# B&R Automation Studio project NAEUL004C00R13L518F00 (part 75)

#### PrecededBySelfBackground1.st
```iecst
ACTION PrecededBySelfBackground1:

	//Converting BA from US Hermes to Rcp
	IF p_bLinkOpsRun THEN
		IF  p_bHermesBADataAccepted THEN
			tyCurrReqRcp.sBoardId := p_tyHermesBARcv.tyData.sBoardId;
			tyCurrReqRcp.sBoardIdCreatedBy := p_tyHermesBARcv.tyData.sBoardIdCreatedBy;
			tyCurrReqRcp.eFailedBoard := p_tyHermesBARcv.tyData.eFailedBoard;
			tyCurrReqRcp.sProductTypeId := p_tyHermesBARcv.tyData.sProductTypeId;
			tyCurrReqRcp.eFlippedBoard := p_tyHermesBARcv.tyData.eFlippedBoard;
			tyCurrReqRcp.sTopBarcode := p_tyHermesBARcv.tyData.sTopBarcode;
			tyCurrReqRcp.sBottomBarcode := p_tyHermesBARcv.tyData.sBottomBarcode;
			tyCurrReqRcp.rLength := p_tyHermesBARcv.tyData.rLength;
			tyCurrReqRcp.rWidth := p_tyHermesBARcv.tyData.rWidth;
			tyCurrReqRcp.rThickness := p_tyHermesBARcv.tyData.rThickness;
			tyCurrReqRcp.rConveyorSpeed := p_tyHermesBARcv.tyData.rConveyorSpeed;
			tyCurrReqRcp.rTopClearanceHeight := p_tyHermesBARcv.tyData.rTopClearanceHeight;
			tyCurrReqRcp.rBottomClearanceHeight := p_tyHermesBARcv.tyData.rBottomClearanceHeight;
			tyCurrReqRcp.rWeight := p_tyHermesBARcv.tyData.rWeight;
			tyCurrReqRcp.sWorkOrderId := p_tyHermesBARcv.tyData.sWorkOrderId;
			tyCurrReqRcp.sBatchId := p_tyHermesBARcv.tyData.sBatchId;
		ELSIF p_bHermesBFDataAccepted THEN
			//Converting BF from US Hermes to Rcp
			tyCurrReqRcp.sBoardId := p_tyHermesBFRcv.tyData.sBoardId;
			tyCurrReqRcp.sBoardIdCreatedBy := p_tyHermesBFRcv.tyData.sBoardIdCreatedBy;
			tyCurrReqRcp.eFailedBoard := p_tyHermesBFRcv.tyData.eFailedBoard;
			tyCurrReqRcp.sProductTypeId := p_tyHermesBFRcv.tyData.sProductTypeId;
			tyCurrReqRcp.eFlippedBoard := p_tyHermesBFRcv.tyData.eFlippedBoard;
			tyCurrReqRcp.sTopBarcode := p_tyHermesBFRcv.tyData.sTopBarcode;
			tyCurrReqRcp.sBottomBarcode := p_tyHermesBFRcv.tyData.sBottomBarcode;
			tyCurrReqRcp.rLength := p_tyHermesBFRcv.tyData.rLength;
			tyCurrReqRcp.rWidth := p_tyHermesBFRcv.tyData.rWidth;
			tyCurrReqRcp.rThickness := p_tyHermesBFRcv.tyData.rThickness;
			tyCurrReqRcp.rConveyorSpeed := p_tyHermesBFRcv.tyData.rConveyorSpeed;
			tyCurrReqRcp.rTopClearanceHeight := p_tyHermesBFRcv.tyData.rTopClearanceHeight;
			tyCurrReqRcp.rBottomClearanceHeight := p_tyHermesBFRcv.tyData.rBottomClearanceHeight;
			tyCurrReqRcp.rWeight := p_tyHermesBFRcv.tyData.rWeight;
			tyCurrReqRcp.sWorkOrderId := p_tyHermesBFRcv.tyData.sWorkOrderId;
			tyCurrReqRcp.sBatchId := p_tyHermesBFRcv.tyData.sBatchId;
		END_IF
	END_IF

	//For Zone 1 Initialization Only
	IF bInitializedFollower1Done = FALSE AND p_bLinkOpsRun THEN
		IF tyCurrZ1Rcp.rWidth = 0 THEN //nothing found in retain
			IF p_bHermesBrdAvlDataNewBrdAvl1stZ  THEN //if no brd retain
				IF p_tyInternalReqProdRcp.diWidthInUM <> 0 THEN
					tyCurrZ1Rcp.rWidth := p_tyInternalReqProdRcp.diWidthInUM/1000 ;
				ELSE //internalReq Rcp=0
					tyCurrZ1Rcp.rWidth := p_diNtParamProdRcpMinWidth/1000 ;
				END_IF
			ELSE //taken From Hermes Retain
				fbParseBrdAvlExternal.p_XMLTable := ADR(pa_tyLinkXMLTableDataBrdAvl1);
				fbParseBrdAvlExternal.iTotalIdxWrite := p_iLinkXMLTableDataBrdAvlTtlIdx1;
				fbParseBrdAvlExternal;

				tyCurrZ1Rcp.sBoardId := fbParseBrdAvlExternal.tyBoardAvailable.tyData.sBoardId;
				tyCurrZ1Rcp.sBoardIdCreatedBy := fbParseBrdAvlExternal.tyBoardAvailable.tyData.sBoardIdCreatedBy;
				tyCurrZ1Rcp.eFailedBoard := fbParseBrdAvlExternal.tyBoardAvailable.tyData.eFailedBoard;
				tyCurrZ1Rcp.sProductTypeId := fbParseBrdAvlExternal.tyBoardAvailable.tyData.sProductTypeId;
				tyCurrZ1Rcp.eFlippedBoard := fbParseBrdAvlExternal.tyBoardAvailable.tyData.eFlippedBoard;
				tyCurrZ1Rcp.sTopBarcode := fbParseBrdAvlExternal.tyBoardAvailable.tyData.sTopBarcode;
				tyCurrZ1Rcp.sBottomBarcode := fbParseBrdAvlExternal.tyBoardAvailable.tyData.sBottomBarcode;
				tyCurrZ1Rcp.rLength := fbParseBrdAvlExternal.tyBoardAvailable.tyData.rLength;
				tyCurrZ1Rcp.rWidth := fbParseBrdAvlExternal.tyBoardAvailable.tyData.rWidth;
				tyCurrZ1Rcp.rThickness := fbParseBrdAvlExternal.tyBoardAvailable.tyData.rThickness;
				tyCurrZ1Rcp.rConveyorSpeed := fbParseBrdAvlExternal.tyBoardAvailable.tyData.rConveyorSpeed;
				tyCurrZ1Rcp.rTopClearanceHeight := fbParseBrdAvlExternal.tyBoardAvailable.tyData.rTopClearanceHeight;
				tyCurrZ1Rcp.rBottomClearanceHeight := fbParseBrdAvlExternal.tyBoardAvailable.tyData.rBottomClearanceHeight;
				tyCurrZ1Rcp.rWeight := fbParseBrdAvlExternal.tyBoardAvailable.tyData.rWeight;
				tyCurrZ1Rcp.sWorkOrderId := fbParseBrdAvlExternal.tyBoardAvailable.tyData.sWorkOrderId;
				tyCurrZ1Rcp.sBatchId := fbParseBrdAvlExternal.tyBoardAvailable.tyData.sBatchId;
			END_IF
		END_IF
		bOverWriteTravLifProperties := TRUE;
		bInitializedFollower1Done := TRUE;
	END_IF

	//Error Handling
	IF p_bLinkOpsRun AND (p_bHermesBADataAccepted OR p_bHermesBFDataAccepted) THEN //
		IF tyCurrReqRcp.rWidth < DINT_TO_REAL(p_diNtParamProdRcpMinWidth)/1000.0 THEN
			eStatus := Error;
			udiStatus := 10010;
		ELSIF tyCurrReqRcp.rWidth  > DINT_TO_REAL(p_diNtParamProdRcpMaxWidth)/1000.0 THEN
			eStatus := Error;
			udiStatus := 10011;
		ELSIF  tyCurrReqRcp.rThickness  > DINT_TO_REAL(p_eNtParamAutoRcpParamLmt.diThicknessInUM)/1000.0 THEN
			eStatus := Error;
			udiStatus := 10012;
		ELSIF  tyCurrReqRcp.rBottomClearanceHeight  > DINT_TO_REAL(p_eNtParamAutoRcpParamLmt.diMaxBottomCleranceInUM)/1000.0 THEN
			eStatus := Error;
			udiStatus := 10013;
		ELSIF tyCurrReqRcp.rTopClearanceHeight > DINT_TO_REAL(p_eNtParamAutoRcpParamLmt.diMaxTopClearamceInUM)/1000.0 THEN
			eStatus := Error;
			udiStatus := 10014;
		END_IF
		IF eStatus = Error THEN
			memset(ADR(tyCurrReqRcp),0,SIZEOF(tyCurrReqRcp));
		END_IF
	END_IF

	IF eStatus <> Error THEN //do not feed F1 with F2 with invalid recipe
		//Follower1
		IF memcmp(ADR(tyCurrZ1Rcp) , ADR(tyCurrReqRcp) , SIZEOF(tyCurrZ1Rcp)) <> 0 AND tyCurrReqRcp.rWidth <> 0 THEN
			bTravLifWidthDiffBlk := TRUE;
			IF p_bZ1AccNewRcpCondition THEN
				tyCurrZ1Rcp := tyCurrReqRcp;
				bOverWriteTravLifProperties := TRUE;
				usiChg2 := usiChg2 +1;
			END_IF
		ELSE
			bTravLifWidthDiffBlk := FALSE;
			bOverWriteTravLifProperties := TRUE;
		END_IF

		//Follower 2
		FOR ii:= 1 TO SIZEOF(a_bBufferMagPresent)/SIZEOF(a_bBufferMagPresent[1]) DO
			IF p_bZ2AccNewRcpCondition THEN	 //in Ops
				IF a_bBufferMagPresent[ii] = FALSE THEN //all time , at the start time
					memset((ADR(a_tyCurrZ2Rcp[1])+(ii-1)*SIZEOF(a_tyCurrZ2Rcp[1])),0,SIZEOF(a_tyCurrZ2Rcp[1])) ;
					a_bMagChangOverBlk[ii] := FALSE;
				ELSE //if present
					p_tyCmpRcp ACCESS (ADR(a_tyCurrZ2Rcp[1])+(ii-1)*SIZEOF(a_tyCurrZ2Rcp[1])) ;
					a_bCheckDifferent[ii]:= (p_tyCmpRcp.sProductTypeId <> tyCurrZ1Rcp.sProductTypeId) OR
					(p_tyCmpRcp.sBatchId <> tyCurrZ1Rcp.sBatchId AND p_bMcParamAutoRcpBatchIDChgCmp) OR
					(p_tyCmpRcp.sWorkOrderId <> tyCurrZ1Rcp.sWorkOrderId) OR
					p_tyCmpRcp.rWidth <> tyCurrZ1Rcp.rWidth OR
					(p_tyCmpRcp.rTopClearanceHeight <> tyCurrZ1Rcp.rTopClearanceHeight AND NOT(p_bMcParamAutoRcpIgnoreTopClr)) OR
					(p_tyCmpRcp.rBottomClearanceHeight <> tyCurrZ1Rcp.rBottomClearanceHeight AND NOT(p_bMcParamAutoRcpIgnoreBtmClr)) OR
					(p_tyCmpRcp.rThickness <> tyCurrZ1Rcp.rThickness AND NOT(p_bMcParamAutoRcpIgnoreThickns)) OR
					p_tyCmpRcp.eFlippedBoard <> tyCurrZ1Rcp.eFlippedBoard	;
					IF a_bCheckDifferent[ii] THEN
						a_bAllwChangeWidth[ii] := FALSE;
						IF a_tyBffrStat[ii].bBffrMty THEN //udiAllwGo and WidthDiff and empty then change rcp
							p_tyCmpRcp := tyCurrZ1Rcp;
							usiChg := usiChg + 1;
							a_bMagChangOverBlk[ii] := FALSE;
							bOverWriteMagProperties := TRUE;
							a_bAllwChangeSlot[ii]  := TRUE;
						ELSE // WidthDiff and not empty then blk
							a_bMagChangOverBlk[ii] := TRUE;
						END_IF
					ELSE //if rcp same mean changewidth allow change until width is same
						a_bMagChangOverBlk[ii] := FALSE;
						a_bAllwChangeWidth[ii] := (a_bMagAWWidthDiff[ii] OR a_bForceChgWidthIfSameRcp[ii]) AND a_tyBffrStat[ii].bBffrMty AND p_bNtParamProjMagAWPrep;

					END_IF

				END_IF

			END_IF
		END_FOR
	END_IF
	//wait new udiAllwGo to toggle and FIND the other empty to change

	//IF all was block with magazine available then Force the Magazine Exit
	iChgOvrCntr := 0;
	FOR ii:= 1 TO SIZEOF(a_bBufferMagPresent)/SIZEOF(a_bBufferMagPresent[1]) DO
		IF  (a_bBufferMagPresent[ii] AND a_bMagChangOverBlk[ii] = TRUE) THEN
			iChgOvrCntr := iChgOvrCntr +1 ;
			EXIT;
		END_IF
	END_FOR
	IF iChgOvrCntr >= 1 THEN
		bForceExitMag := TRUE; //force Magazine to exit the highest priority Mag
	ELSE
		bForceExitMag := FALSE;
	END_IF

END_ACTION
```

#### PrecededBySelfBackground2.st
```iecst
ACTION PrecededBySelfBackground2:

	//Convert ProdID to Rcp Name and rWidth to diWidth for F0 to output Hermes
	sProdtypeID:= tyCurrReqRcp.sProductTypeId;
	diProdWidth := REAL_TO_DINT(tyCurrReqRcp.rWidth*1000);

	//Convert to Width for F1
	IF bOverWriteTravLifProperties THEN
		diTravLifWidth := REAL_TO_DINT(tyCurrZ1Rcp.rWidth*1000);
		bOverWriteTravLifProperties	:= FALSE;
	END_IF

	//Convert to Pitch for F2
	IF bOverWriteMagProperties = TRUE THEN
		//overwriting diMax
		FOR kk := 1 TO SIZEOF(a_tyCurrZ2Rcp)/SIZEOF(a_tyCurrZ2Rcp[1]) DO
			p_diRequestedMinSlt := 3;
			p_diRequestedGapToMaxSlt := 0;
			IF p_bProdRcp0ToptoBtm THEN
				IF p_diRequestedGapToMaxSlt > ((a_tyCurrZ2Rcp[kk].rTopClearanceHeight + a_tyCurrZ2Rcp[kk].rThickness)/(p_diMagRcpCurrRcpSltToSlt/1000)) THEN
					rMaxslt := (p_diMagRcpCurrRcpTtlSlt-p_diRequestedGapToMaxSlt)  ;
				ELSE
					rMaxslt := p_diMagRcpCurrRcpTtlSlt - ((a_tyCurrZ2Rcp[kk].rTopClearanceHeight + a_tyCurrZ2Rcp[kk].rThickness)/(p_diMagRcpCurrRcpSltToSlt/1000)) + 1;
				END_IF
				rMinslt :=  (a_tyCurrZ2Rcp[kk].rBottomClearanceHeight)/(p_diMagRcpCurrRcpSltToSlt/1000);
				rPitch := (a_tyCurrZ2Rcp[kk].rTopClearanceHeight + a_tyCurrZ2Rcp[kk].rBottomClearanceHeight + a_tyCurrZ2Rcp[kk].rThickness)/(p_diMagRcpCurrRcpSltToSlt/1000);
				IF rPitch = 0 THEN
					rPitch := 1;
				END_IF
				rNumInterval := (rMaxslt - rMinslt )/ceil(rPitch);
				diCalcedMax := REAL_TO_DINT(floor(rMaxslt));
				diCalcedPitch := REAL_TO_DINT(ceil(rPitch));
				diCalcedMin := REAL_TO_DINT((diCalcedMax - floor(rNumInterval)*ceil(rPitch)));

				IF diCalcedMin = 0 THEN
					diCalcedMin := diCalcedPitch;
				END_IF

			ELSE
				IF p_diRequestedMinSlt = 0 THEN
					p_diRequestedMinSlt := 1;
				END_IF
				IF ceil((a_tyCurrZ2Rcp[kk].rBottomClearanceHeight)/(p_diMagRcpCurrRcpSltToSlt/1000)) >= p_diRequestedMinSlt THEN
					rMinslt := (a_tyCurrZ2Rcp[kk].rBottomClearanceHeight)/(p_diMagRcpCurrRcpSltToSlt/1000) + 1;
				ELSE
					rMinslt :=  p_diRequestedMinSlt;
				END_IF
				//+ (a_tyCurrZ2Rcp[kk].rBottomClearanceHeight)/(p_diMagRcpCurrRcpSltToSlt/1000);
				rMaxslt := p_diMagRcpCurrRcpTtlSlt-((a_tyCurrZ2Rcp[kk].rTopClearanceHeight + a_tyCurrZ2Rcp[kk].rThickness)/(p_diMagRcpCurrRcpSltToSlt/1000)) +1;
				rPitch := (a_tyCurrZ2Rcp[kk].rTopClearanceHeight + a_tyCurrZ2Rcp[kk].rBottomClearanceHeight + a_tyCurrZ2Rcp[kk].rThickness)/(p_diMagRcpCurrRcpSltToSlt/1000);
				IF rPitch = 0 THEN
					rPitch := 1;
				END_IF
				rNumInterval := (rMaxslt - rMinslt )/ceil(rPitch);
				diCalcedMin := REAL_TO_DINT(ceil(rMinslt));
				diCalcedPitch := REAL_TO_DINT(ceil(rPitch));
				diCalcedMax := REAL_TO_DINT((diCalcedMin + floor(rNumInterval)*ceil(rPitch)));

				IF diCalcedMax = p_diMagRcpCurrRcpTtlSlt + 1 THEN
					diCalcedMax := diCalcedMax - diCalcedPitch;
				END_IF

			END_IF
			a_tyMagProps[kk].diMaxSlt := diCalcedMax;
			a_tyMagProps[kk].diMinSlt := diCalcedMin;
			a_tyMagProps[kk].diPitch  := diCalcedPitch;
			a_tyMagProps[kk].diWidth := REAL_TO_DINT(a_tyCurrZ2Rcp[kk].rWidth * 1000);
		END_FOR

		bOverWriteMagProperties := FALSE;
	END_IF

	//			IF diCalcedMin < p_diRequestedMinSlt THEN
	//				diModulus :=  p_diRequestedMinSlt/diCalcedMin;
	//				diCalcedMin := diCalcedMin + diModulus*diCalcedPitch;
	//			END_IF
END_ACTION
```

#### Package Logical/AutoRcp/AutoRcp/PrecededByF1 - Intended for F2 only

#### PrecededByF1Initial.st
```iecst
ACTION PrecededByF1Initial:

	//Mag Detail (Rcp)
	fbFileRead1.sDevice			:= 'Retain';
	fbFileRead1.sFile			:= 'MagazinePropsRcp';
	fbFileRead1.udiOffset		:= 0;
	fbFileRead1.p_Dest			:= ADR(a_tyMagProps);
	fbFileRead1.udiLen			:= SIZEOF(a_tyMagProps);
	fbFileRead1(bEn := FALSE);

	fbFileWrite1.sDevice	:= 'Retain';
	fbFileWrite1.sFile			:= 'MagazinePropsRcp';
	fbFileWrite1.udiOffset		:= 0;
	fbFileWrite1.p_Src			:= ADR(a_tyMagPropsWr);
	fbFileWrite1.udiLen			:= SIZEOF(a_tyMagPropsWr);
	fbFileWrite1.udiOption		:= 0;
	fbFileWrite1(bEn := FALSE);

	//artibitrary type  on Zone 1 (Traverser)
	IF p_bNtParamF1ArbitraryType THEN
		fbFileRead2.sDevice			:= 'Retain';
		fbFileRead2.sFile			:= 'TravRcp';
		fbFileRead2.udiOffset		:= 0;
		fbFileRead2.p_Dest			:= ADR(tyCurrZ1Rcp);
		fbFileRead2.udiLen			:= SIZEOF(tyCurrZ1Rcp);
		fbFileRead2(bEn := FALSE);

		fbFileWrite2.sDevice	:= 'Retain';
		fbFileWrite2.sFile			:= 'TravRcp';
		fbFileWrite2.udiOffset		:= 0;
		fbFileWrite2.p_Src			:= ADR(tyZ1RcpWr);
		fbFileWrite2.udiLen			:= SIZEOF(tyZ1RcpWr);
		fbFileWrite2.udiOption		:= 0;
		fbFileWrite2(bEn := FALSE);
	END_IF
END_ACTION
```

#### PrecededByF1Link.st
```iecst
ACTION PrecededByF1Link:

	p_bZ2AccNewRcpCondition := (p_bLinkOpsRun = TRUE);// AND (p_bLinkOpsMagConvUL1InitDone AND p_bLinkOpsMagConvUL2InitDone AND p_bLinkOpsMagConvUL3InitDone);

	IF p_bNtParamF1ArbitraryType THEN
		p_bZ1AccNewRcpCondition := (p_bLinkOpsRun = TRUE) AND (p_bLinkOpsTravLifULInitDone = TRUE) AND (p_bLinkPshrConvHvBrd = TRUE);

		IF p_sTCPBtmFullMsgRd <> '' THEN
			tyCurrReqRcp.sBottomBarcode := p_sTCPBtmFullMsgRd;
		END_IF
	END_IF

END_ACTION
```

#### PrecededByF1Background1.st
```iecst
ACTION PrecededByF1Background1:
	//Requesting
	IF NOT(p_bNtParamF1ArbitraryType) THEN //F1 Rcp compare
		tyCurrReqMagRcp.diMaxSlt := p_tyInternalReqProdRcp.diMaxSltValue;
		tyCurrReqMagRcp.diMinSlt := p_tyInternalReqProdRcp.diMinSltValue;
		tyCurrReqMagRcp.diPitch  := p_tyInternalReqProdRcp.diPitch;
		tyCurrReqMagRcp.diWidth  := p_tyInternalReqProdRcp.diWidthInUM;
		tyCurrReqMagRcp.sRcpNm   := p_tyInternalReqProdRcp.sRcpNm;
	ELSE
		//artibitrary type
		IF memcmp(ADR(tyCurrZ1Rcp) , ADR(tyCurrReqRcp) , SIZEOF(tyCurrZ1Rcp)) <> 0 AND (tyCurrReqRcp.rWidth <> 0 OR p_bNtParamF1ArbitraryType) THEN
			IF p_bZ1AccNewRcpCondition THEN
				tyCurrZ1Rcp := tyCurrReqRcp;
				bOverWriteTravLifProperties := TRUE;
				usiChg2 := usiChg2 +1;
			END_IF
		END_IF
		tyCurrReqMagRcp.sTrailingBarcode := RIGHT(tyCurrZ1Rcp.sBottomBarcode,10);//length of comparision
	END_IF

	//Follower 2
	FOR ii:= 1 TO SIZEOF(a_bBufferMagPresent)/SIZEOF(a_bBufferMagPresent[1]) DO
		IF p_bZ2AccNewRcpCondition THEN	 //in Ops
			IF a_bBufferMagPresent[ii] = FALSE THEN //all time , at the start time
				memset((ADR(a_tyMagProps[1])+(ii-1)*SIZEOF(a_tyMagProps[1])),0,SIZEOF(a_tyMagProps[1])) ;
				a_bMagChangOverBlk[ii] := FALSE;
			ELSE //if present
				p_tyMagCmpRcp ACCESS (ADR(a_tyMagProps[1])+(ii-1)*SIZEOF(a_tyMagProps[1])) ;
				a_bCheckDifferent[ii] := (memcmp(ADR(p_tyMagCmpRcp),ADR(tyCurrReqMagRcp),SIZEOF(p_tyMagCmpRcp)) <> 0) AND (tyCurrReqMagRcp.diWidth <> 0 OR p_bNtParamF1ArbitraryType);
				IF a_bCheckDifferent[ii] THEN
					a_bAllwChangeWidth[ii] := FALSE;
					IF a_tyBffrStat[ii].bBffrMty THEN //udiAllwGo and WidthDiff and empty then change rcp
						p_tyMagCmpRcp := tyCurrReqMagRcp;
						usiChg := usiChg + 1;
						a_bMagChangOverBlk[ii] := FALSE;
						bOverWriteMagProperties := TRUE;
						a_bAllwChangeSlot[ii]  := TRUE;
					ELSE // WidthDiff and not empty then blk
						a_bMagChangOverBlk[ii] := TRUE;
					END_IF
				ELSE //if rcp same mean changewidth allow change until width is same
					a_bMagChangOverBlk[ii] := FALSE;
					a_bAllwChangeWidth[ii] := (a_bMagAWWidthDiff[ii] OR a_bForceChgWidthIfSameRcp[ii]) AND a_tyBffrStat[ii].bBffrMty AND p_bNtParamProjMagAWPrep;
				END_IF

			END_IF
		END_IF
	END_FOR

END_ACTION
```

#### PrecededByF1Background2.st
```iecst
ACTION PrecededByF1Background2:

END_ACTION
```

#### Init.st - Change By Project
```iecst
(** 2019-06-27 **)
PROGRAM _INIT

	(* Always Change If Project Change *)

	//Physical Configuration
	bAutoUpdtData	:= TRUE;
	bInternalUse	:= TRUE;

	//Pass Address To Global Address For External Use
	//Action, State & Status
	p_AutoRcpStat		:= ADR(eStat);
	p_AutoRcpStatus	:= ADR(eStatus);

	//Alarm
	p_AutoRcpAlmData		:= ADR(tyAlmData);
	p_AutoRcpInfoData		:= ADR(tyInfoData);
	p_AutoRcpInfoData1	:= ADR(tyInfoData1);

	//Output
//	p_AutoRcpUSAllow			:= ADR(bUSAllow);
//	p_AutoRcpDSAllow			:= ADR(bDSAllow);

	p_AutoRcpCurrRcpProdID	:= ADR(sProdtypeID);
	p_AutoRcpCurrRcpWidth :=  ADR(diProdWidth);

	p_AutoRcpbTravWidthDiffblk := ADR(bTravLifWidthDiffBlk);

	(*p_AutoRcp:= ADR(a_bCheckDifferent);*)
	p_AutoRcpbMag1PropDiffBlk := ADR(a_bCheckDifferent[1]);
	p_AutoRcpbMag2PropDiffBlk := ADR(a_bCheckDifferent[2]);
	p_AutoRcpbMag3PropDiffBlk := ADR(a_bCheckDifferent[3]);

	p_AutoRcpbMagChangeOverBlk := ADR(a_bMagChangOverBlk);

	p_AutoRcpbMag1WidthChg	:= ADR (a_bAllwChangeWidth[1]);
	p_AutoRcpbMag2WidthChg	:= ADR (a_bAllwChangeWidth[2]);
	p_AutoRcpbMag3WidthChg	:= ADR (a_bAllwChangeWidth[3]);

	p_AutoRcpbMag1SlotChg := ADR (a_bAllwChangeSlot[1]);
	p_AutoRcpbMag2SlotChg := ADR (a_bAllwChangeSlot[2]);
	p_AutoRcpbMag3SlotChg := ADR (a_bAllwChangeSlot[3]);

	p_diAutoRcpTravLifWidth := ADR(diTravLifWidth);

	p_diAutoRcpAllMagProps := ADR(a_tyMagProps);
	p_diAutoRcpBrdProps    := ADR(a_tyCurrZ2Rcp);

	p_diAutoRcpMag1MaxSlt  := ADR(a_tyMagProps[1].diMaxSlt);
	p_diAutoRcpMag1MinSlt  := ADR(a_tyMagProps[1].diMinSlt);
	p_diAutoRcpMag1Pitch   := ADR(a_tyMagProps[1].diPitch);
	p_diAutoRcpMag1Width   := ADR(a_tyMagProps[1].diWidth);

	p_diAutoRcpMag2MaxSlt  := ADR(a_tyMagProps[2].diMaxSlt);
	p_diAutoRcpMag2MinSlt  := ADR(a_tyMagProps[2].diMinSlt);
	p_diAutoRcpMag2Pitch   := ADR(a_tyMagProps[2].diPitch);
	p_diAutoRcpMag2Width   := ADR(a_tyMagProps[2].diWidth);

	p_diAutoRcpMag3MaxSlt  := ADR(a_tyMagProps[3].diMaxSlt);
	p_diAutoRcpMag3MinSlt  := ADR(a_tyMagProps[3].diMinSlt);
	p_diAutoRcpMag3Pitch   := ADR(a_tyMagProps[3].diPitch);
	p_diAutoRcpMag3Width   := ADR(a_tyMagProps[3].diWidth);

	p_AutoRcpForceExitMag		   := ADR(bForceExitMag);
	(* Always Change If Project Change *)

END_PROGRAM
```

#### Act_InitGlobal.st - Change By Project
```iecst
(** 2019-06-12 **)
ACTION Act_InitGlobal:

	(* Always Change If Project Change *)

	//Pass Data To Link
	p_bLinkStartupRun ACCESS p_StartupRun;

	p_bLinkOpsRun ACCESS p_OpsRun;
	p_eLinkNtParamProjMag ACCESS p_NtParamProjMag;

	//Pass Data To Internal Use
	p_udiRstErr ACCESS p_RstErrReset;
	//p_tyInternalReqProdRcp ACCESS p_Follower1UpdtProdRcp;	//Follower 2 Assign With Follower 1 Recipe
	p_sProgNm ACCESS p_NtParamAutoRcpProgNm;
	p_bNtSettingsLoadDone ACCESS p_StartupNtSettingsLoadDone;

	p_bNtParamAutoRcpPrep ACCESS p_NtParamAutoRcpPrep;
	p_bMcParamAutoRcpDis  ACCESS p_McParamAutoRcpDisable;
	//Zone 1
	p_bLinkPshrConvHvBrd ACCESS p_PshrConvHvBrd;
	p_bLinkOpsTravLifULInitDone ACCESS p_OpsTravLifULInitDone;

	//Zone 2
	p_bLinkOpsMagConvUL1InitDone ACCESS p_OpsMagConvUL1InitDone;
	p_bLinkOpsMagConvUL2InitDone ACCESS p_OpsMagConvUL2InitDone;
	p_bLinkOpsMagConvUL3InitDone ACCESS p_OpsMagConvUL3InitDone;
	p_udiOpsMagConvUL1MagAllwGo ACCESS p_OpsMagConvUL1MagAllwGo;
	p_udiOpsMagConvUL2MagAllwGo ACCESS p_OpsMagConvUL2MagAllwGo;
	p_udiOpsMagConvUL3MagAllwGo ACCESS p_OpsMagConvUL3MagAllwGo;

	p_bBuffer1MagPresent ACCESS p_Buffer1MagPresent;
	p_bBuffer2MagPresent ACCESS p_Buffer2MagPresent;
	p_bBuffer3MagPresent ACCESS p_Buffer3MagPresent;

	p_bBuffer1MagRemoved ACCESS p_Buffer1MagPresent;
	p_bBuffer2MagRemoved ACCESS p_Buffer2MagPresent;
	p_bBuffer3MagRemoved ACCESS p_Buffer3MagPresent;

	p_tyBuffer1BffrStat ACCESS p_Buffer1BffrStat ;
	p_tyBuffer2BffrStat ACCESS p_Buffer2BffrStat ;
	p_tyBuffer3BffrStat ACCESS p_Buffer3BffrStat ;

	p_bMagAW1WidthDiff ACCESS p_MagAWOpen1WidthPosDiff;
	p_bMagAW2WidthDiff ACCESS p_MagAWOpen2WidthPosDiff;
	p_bMagAW3WidthDiff ACCESS p_MagAWOpen3WidthPosDiff;

	//Hermes A accepted the BA
	p_bHermesABAAccepted ACCESS p_USHermesABAAccepted;
	p_bHermesABFAccepted ACCESS p_USHermesABFAccepted;

	//Hermes B accepeted the BA
	p_bHermesBBAAccepted ACCESS p_USHermesBBAAccepted;
	p_bHermesBBFAccepted ACCESS p_USHermesBBFAccepted;

	p_diMagRcpCurrRcpTtlSlt ACCESS p_MagRcpCurrRcpTtlSlt;
	p_diMagRcpCurrRcpSltToSlt ACCESS p_MagRcpCurrRcpSltToSlt;

	//p_tyInternalReqProdRcp ACCESS p_ProdRcpCurrRcp0;
	p_bProdRcp0ToptoBtm ACCESS p_ProdRcpCurrRcp0TopToBtm;
	//for Board Retain
	p_bHermesBrdAvlDataNewBrdAvl1stZ ACCESS p_HermesBrdAvlDataNewBrdAvl1stZ;
	pa_tyLinkXMLTableDataBrdAvl1 ACCESS p_HermesBrdAvlDataTable1stZ; //lane 1 B.A
	p_iLinkXMLTableDataBrdAvlTtlIdx1 ACCESS p_HermesBrdAvlDataTtlIdx1stZ; //lane 1 B.A

	p_usiLinkProdRcpCurrRcpMcMod ACCESS p_ProdRcpCurrRcp0McMod;
	pa_bMagRej ACCESS p_OpsTravLifULMagRej;

	p_bOpsMagConvUL1AWDone ACCESS p_OpsMagConvUL1AWDone; //to froce AW
	p_bOpsMagConvUL2AWDone ACCESS p_OpsMagConvUL2AWDone;
	p_bOpsMagConvUL3AWDone ACCESS p_OpsMagConvUL3AWDone;

	p_bOpsMagConvUL1SlotUpdtDone ACCESS p_OpsMagConvUL1SlotUpdtDone; //to update pitch
	p_bOpsMagConvUL2SlotUpdtDone ACCESS  p_OpsMagConvUL2SlotUpdtDone;
	p_bOpsMagConvUL3SlotUpdtDone ACCESS p_OpsMagConvUL3SlotUpdtDone;
	p_bMcParamAutoRcpBatchIDChgCmp	ACCESS p_McParamAutoRcpBatchIDChgCmp;
	p_bMcParamAutoRcpIgnoreBtmClr ACCESS p_McParamAutoRcpIgnoreBtmClr;
	p_bMcParamAutoRcpIgnoreTopClr ACCESS p_McParamAutoRcpIgnoreTopClr;
	p_bMcParamAutoRcpIgnoreThickns ACCESS p_McParamAutoRcpIgnoreThickns;

	//Error Handling Parameter
	p_eNtParamAutoRcpParamLmt ACCESS p_NtParamAutoRcpParamLmt;
	p_diNtParamProdRcpMinWidth ACCESS p_NtParamProdRcpMinWidth;
	p_diNtParamProdRcpMaxWidth ACCESS p_NtParamProdRcpMaxWidth;

	//We Fab

	p_tyInternalReqProdRcp ACCESS p_Follower1UpdtProdRcp;	//Follower 2 Assign With Follower 1 Recipe
	p_eNtParamAutoRcpPrecededBy ACCESS p_NtParamAutoRcpPrecededBy;

	//Mag AW Prep
	p_bNtParamProjMagAWPrep ACCESS p_NtParamProjMagAWPrep;

	//Adding Arbitrary type for Flushing Magazine
	p_bNtParamF1ArbitraryType ACCESS p_NtParamAutoRcpF1ArbitraryType;

	p_sTCPBtmFullMsgRd ACCESS p_TCPBtmFullMsgRd;
	p_sTCPTopFullMsgRd ACCESS p_TCPTopFullMsgRd;
END_ACTION
```

#### InputRef_Link.var - Change By Project
```iecst
(*2019-05-07*)
(**)
VAR
	p_bLinkStartupRun : REFERENCE TO BOOL;
END_VAR
(**)
VAR
	p_bLinkOpsRun : REFERENCE TO BOOL;
	p_eLinkNtParamProjMag : REFERENCE TO eULMag;
	p_bLinkPshrConvHvBrd : REFERENCE TO BOOL;
	p_bLinkOpsTravLifULInitDone : REFERENCE TO BOOL;
	p_bLinkMagConvInitDone : BOOL;
	p_bLinkNtParamProjMagConv1Prep : REFERENCE TO BOOL;
	p_bLinkNtParamProjMagConv2Prep : REFERENCE TO BOOL;
	p_bLinkNtParamProjMagConv3Prep : REFERENCE TO BOOL;
	p_bLinkBffr1MagRemoved : REFERENCE TO BOOL;
	p_bLinkBffr2MagRemoved : REFERENCE TO BOOL;
	p_bLinkBffr3MagRemoved : REFERENCE TO BOOL;
	p_bLinkOpsMagUL1InitDone : REFERENCE TO BOOL;
	p_bLinkOpsMagUL2InitDone : REFERENCE TO BOOL;
	p_bLinkOpsMagUL3InitDone : REFERENCE TO BOOL;
	p_bLinkOpsMagConvUL1InitDone : REFERENCE TO BOOL;
	p_bLinkOpsMagConvUL2InitDone : REFERENCE TO BOOL;
	p_bLinkOpsMagConvUL3InitDone : REFERENCE TO BOOL;
	p_tyBuffer1BffrStat : REFERENCE TO tyBffrStat;
	p_tyBuffer2BffrStat : REFERENCE TO tyBffrStat;
	p_tyBuffer3BffrStat : REFERENCE TO tyBffrStat;
	p_bMagAW1WidthDiff : REFERENCE TO BOOL;
	p_bMagAW2WidthDiff : REFERENCE TO BOOL;
	p_bMagAW3WidthDiff : REFERENCE TO BOOL;
	p_udiOpsMagConvUL1MagAllwGo : REFERENCE TO UDINT;
	p_udiOpsMagConvUL2MagAllwGo : REFERENCE TO UDINT;
	p_udiOpsMagConvUL3MagAllwGo : REFERENCE TO UDINT;
	p_bZ1AccNewRcpCondition : REFERENCE TO BOOL;
	p_bZ2AccNewRcpCondition : REFERENCE TO BOOL;
	p_diRequestedMinSlt : REFERENCE TO DINT;
	p_diRequestedGapToMaxSlt : REFERENCE TO DINT;
	p_bHermesBADataAccepted : REFERENCE TO BOOL;
	p_bHermesBFDataAccepted : REFERENCE TO BOOL;
	p_bHermesBBAAccepted : REFERENCE TO BOOL;
	p_bHermesABAAccepted : REFERENCE TO BOOL;
	p_bHermesBBFAccepted : REFERENCE TO BOOL;
	p_bHermesABFAccepted : REFERENCE TO BOOL;
	p_tyHermesBARcv : REFERENCE TO tyHermesBoardAvailable;
	p_tyHermesBFRcv : REFERENCE TO tyHermesBoardForecast;
	p_diMagRcpCurrRcpSltToSlt : REFERENCE TO DINT;
	p_diMagRcpCurrRcpTtlSlt : REFERENCE TO DINT;
	p_bBuffer1MagPresent : REFERENCE TO BOOL;
	p_bBuffer2MagPresent : REFERENCE TO BOOL;
	p_bBuffer3MagPresent : REFERENCE TO BOOL;
	p_bBuffer1MagRemoved : REFERENCE TO BOOL;
	p_bBuffer2MagRemoved : REFERENCE TO BOOL;
	p_bBuffer3MagRemoved : REFERENCE TO BOOL;
END_VAR
(**)
VAR
	bOpsInitDone : BOOL;
	p_eLinkUIProdRcpAct : REFERENCE TO eProdRcpAction;
	p_eProdRcpStat : REFERENCE TO eProdRcpAction;
	p_eProdRcpStatus : REFERENCE TO eFBStatus;
	p_tyProdRcpCurrRcpWr : REFERENCE TO tyProdRcpParam;
END_VAR
```

#### Act_LinkAction.st - Change By Project
```iecst
(** 2021-08-01 **)
ACTION Act_LinkAction:

	IF p_bLinkStartupRun = TRUE THEN
		p_eAct ACCESS p_StartupAutoRcpsAct;
	ELSE
		p_eAct ACCESS ADR(eAct);
	END_IF

END_ACTION
```

#### Act_LinkEn.st - Change By Project
```iecst
(** 2019-04-26 **)
ACTION Act_LinkEn:

	//Link bPrep, bEn & bDis
	//p_bDis	:= (p_bLinkStartupRun = TRUE);
	p_bPrep	:= p_bNtParamAutoRcpPrep AND NOT(p_bMcParamAutoRcpDis);

END_ACTION
```

#### Act_Link.st - Change By Project
```iecst
(** 2019-07-04 **)
ACTION Act_Link:

	CASE p_eNtParamAutoRcpPrecededBy OF
		PrecededBySelf:
			PrecededBySelfLink;
		PrecededByF1:
			PrecededByF1Link;
	END_CASE

	//for comparing Rcp
	a_tyBffrStat[1] := p_tyBuffer1BffrStat;
	a_tyBffrStat[2] := p_tyBuffer2BffrStat;
	a_tyBffrStat[3] := p_tyBuffer3BffrStat;

	a_udiMagAllwGo[1] := p_udiOpsMagConvUL1MagAllwGo;
	a_udiMagAllwGo[2] := p_udiOpsMagConvUL2MagAllwGo;
	a_udiMagAllwGo[3] := p_udiOpsMagConvUL3MagAllwGo;

	a_bBufferMagPresent[1] := p_bBuffer1MagPresent; //AND p_bBuffer1MagRemoved = FALSE;
	a_bBufferMagPresent[2] := p_bBuffer2MagPresent; //AND p_bBuffer2MagRemoved = FALSE;
	a_bBufferMagPresent[3] := p_bBuffer3MagPresent;// AND p_bBuffer3MagRemoved = FALSE;

	a_bMagAWWidthDiff[1] := p_bMagAW1WidthDiff;
	a_bMagAWWidthDiff[2] := p_bMagAW2WidthDiff;
	a_bMagAWWidthDiff[3] := p_bMagAW3WidthDiff;

	FOR x:= 1 TO SIZEOF(a_bBufferMagPresent)/SIZEOF(a_bBufferMagPresent[1]) DO
	  	//Force a New Mag with Same Rcp to Chg Width
		IF a_bMagAWWidthDiff[x] = FALSE AND NOT(a_bBufferMagPresent[x]) THEN
			a_bForceChgWidthIfSameRcp[x] := TRUE;
		ELSIF (a_bBufferMagPresent[x]) THEN
			IF p_bOpsMagConvUL1AWDone AND x = 1 THEN
				a_bForceChgWidthIfSameRcp[x] := FALSE;
			ELSIF p_bOpsMagConvUL2AWDone AND x = 2 THEN
				a_bForceChgWidthIfSameRcp[x] := FALSE;
			ELSIF p_bOpsMagConvUL3AWDone AND x = 3 THEN
				a_bForceChgWidthIfSameRcp[x] := FALSE;
			END_IF
		END_IF

	END_FOR

	//Change Completed FeedBack
	IF p_bOpsMagConvUL1SlotUpdtDone THEN
		a_bAllwChangeSlot[1] := FALSE;
	END_IF
	IF p_bOpsMagConvUL2SlotUpdtDone THEN
		a_bAllwChangeSlot[2] := FALSE;
	END_IF
	IF p_bOpsMagConvUL3SlotUpdtDone THEN
		a_bAllwChangeSlot[3] := FALSE;
	END_IF

	p_eULMod	:= USINT_TO_UDINT(p_usiLinkProdRcpCurrRcpMcMod); // 0 Unloader , 1 Rej
END_ACTION
```

#### Cyclic.st - Do Not Change!!!
```iecst
(** 2019-04-21 **)
PROGRAM _CYCLIC

	IF bInitDone = FALSE THEN
		bInitDone	:= TRUE;

		Act_InitLocal;
		Act_InitGlobal;

	ELSIF bInitialDone = FALSE THEN
		IF p_bNtSettingsLoadDone = TRUE THEN
			bInitialDone	:= TRUE;

			Act_Initial;
		END_IF

	ELSE

		Act_RstErr;
		Act_LinkAction;
		Act_Action;
		Act_LinkEn;

		IF (p_bPrep = TRUE) AND (p_bEn = TRUE) AND (p_bDis = FALSE) THEN
			Act_Link;
			Act_Main;
			Act_Background;
			Act_Background2;
		ELSE
			Act_Main_Disable;

		END_IF

		Act_Alarm;

	END_IF

END_PROGRAM
```

#### Act_InitLocal.st - Do Not Change!!!
```iecst
(** 2020-08-06 **)
ACTION Act_InitLocal:

	//Input Reference Link To Local Variable
	p_udiRstErr ACCESS ADR(udiRstErr);
	p_bPrep ACCESS ADR(bPrep);
	p_bEn ACCESS ADR(bEn);
	p_bDis ACCESS ADR(bDis);
	p_sIPAddr ACCESS ADR(sIPAddr);
	p_sMcNm ACCESS ADR(sMcNm);
	p_bAWPrep ACCESS ADR(bAWPrep);
	p_bAWDis ACCESS ADR(bAWDis);
	p_bMnlAccData ACCESS ADR(bMnlAccData);
	p_bSectionLeader ACCESS ADR(bSectionLeader);
	p_sMagRcpNm ACCESS ADR(sMagRcpNm);
	p_diWidthLimit ACCESS ADR(diWidthLimit);
	p_bUSWidthChkPrep ACCESS ADR(bUSWidthChkPrep);
	p_bUSWidthChkEn ACCESS ADR(bUSWidthChkEn);
	p_bUSWidthChkSen ACCESS ADR(bUSWidthChkSen);
	p_bDSWidthChkPrep ACCESS ADR(bDSWidthChkPrep);
	p_bDSWidthChkEn ACCESS ADR(bDSWidthChkEn);
	p_bDSWidthChkSen ACCESS ADR(bDSWidthChkSen);
	p_bProdWidthChk ACCESS ADR(bProdWidthChk);
	p_bUIProdAccData ACCESS ADR(bUIProdAccData);
	p_bUIProdUpdtData ACCESS ADR(bUIProdUpdtData);
	p_bUIMagAccData ACCESS ADR(bUIMagAccData);

	p_tyCmpRcp ACCESS ADR(tyCurrProdRcp);
	p_sCurrMagRcpNm ACCESS ADR(sCurrMagRcpNm);
	p_eTimeStat ACCESS ADR(eTimeStat);
	p_eTimeStatus ACCESS ADR(eTimeStatus);
	p_bAccNewRcpCond ACCESS ADR(bAccNewRcpCond);
	p_bUpdtNewRcpCond ACCESS ADR(bUpdtNewRcpCond);
	p_bAutoUpdtData ACCESS ADR(bAutoUpdtData);
	p_sInfoMsg ACCESS ADR(sInfoMsg);
	p_bInternalUse ACCESS ADR(bInternalUse);
	p_tyInternalReqProdRcp ACCESS ADR(tyInternalReqProdRcp);
	p_bNewBrdEnteredCond ACCESS ADR(bNewBrdEnteredCond);
	p_bOldBrdExitedCond ACCESS ADR(bOldBrdExitedCond);
	p_bRlsBrd ACCESS ADR(bRlsBrd);
	p_tyToLeaderProdRcp ACCESS ADR(tyToLeaderProdRcp);
	pa_bInternalReqProdRcpDiff ACCESS ADR(a_bInternalReqProdRcpDiff);
	p_bUpdtProdRcpDiff ACCESS ADR(bUpdtProdRcpDiff);
	p_bRlsBrdProdRcpDiff ACCESS ADR(bRlsBrdProdRcpDiff);
	p_sProgNm ACCESS ADR(sProgNm);
	p_bNtSettingsLoadDone ACCESS ADR(bNtSettingsLoadDone);
	p_tOnlineChkDlyTm ACCESS ADR(tOnlineChkDlyTm);
	p_bManual ACCESS ADR(bManual);
	p_bErr ACCESS ADR(bErr);
	p_bWarning ACCESS ADR(bWarning);
	p_bOps ACCESS ADR(bOps);
	p_bStandby ACCESS ADR(bStandby);
	p_eAWStat ACCESS ADR(eAWStat);
	p_bWidth2Prep ACCESS ADR(bWidth2Prep);
	p_bDBAOnWOAlign ACCESS ADR(bDBAOnWOAlign);
	p_tyProdRcpCurrRcpWr ACCESS ADR(bDBAOnWOAlign);
	p_eLinkUIProdRcpAct ACCESS ADR(bDBAOnWOAlign);

	p_bZ1AccNewRcpCondition ACCESS ADR(bZ1AccNewRcpCondition);
	p_bZ2AccNewRcpCondition ACCESS ADR(bZ2AccNewRcpCondition);
	p_tyHermesBARcv ACCESS ADR(tyHermesBAAccpt);
	p_tyHermesBFRcv ACCESS ADR(tyHermesBFAccpt);
	p_bHermesBADataAccepted ACCESS  ADR(bHermesBAAccpt);
	p_bHermesBFDataAccepted ACCESS  ADR(bHermesBFAccpt);
	p_diRequestedMinSlt ACCESS ADR(diRequestedMinSlt);
	p_diRequestedGapToMaxSlt ACCESS ADR(diRequestedGapToMaxSlt);

	p_eULMod ACCESS ADR(eULMode);
END_ACTION
```

#### Act_Initial.st - Do Not Change!!!
```iecst
(** 2020-08-06 **)
ACTION Act_Initial:
	fbDirCreate1.sDevice	:= 'F';
	fbDirCreate1.sDirName	:= 'User';
	fbDirCreate1(bEn := FALSE);

	fbDirCreate2.sDevice	:= 'User';
	fbDirCreate2.sDirName	:= 'Retain';
	fbDirCreate2(bEn := FALSE);

	CASE p_eNtParamAutoRcpPrecededBy OF
		PrecededBySelf:
			PrecededBySelfInitial;
		PrecededByF1:
			PrecededByF1Initial;
	END_CASE

END_ACTION
```

#### Act_Background.st - Do Not Change!!!
```iecst
(** 2021-05-18 **)
ACTION Act_Background:

	CASE p_eNtParamAutoRcpPrecededBy OF
		PrecededBySelf:
			PrecededBySelfBackground1;
		PrecededByF1:
			PrecededByF1Background1;
	END_CASE

	//if Trav different, write one time
	IF usiPrevChg2 <> usiChg2
		AND (eStatus = Idle AND eStat = AutoRcpActIdle)  THEN
		tyZ1RcpWr := tyCurrZ1Rcp;
		p_eAct := AutoRcpActWriteRetain2;
	END_IF
	IF eStatus = Done AND eStat = AutoRcpActWriteRetain2 THEN
		usiPrevChg2 :=  usiChg2;
		p_eAct := AutoRcpActIdle;
	END_IF

	//if Mag different, write one time
	IF usiPrevChg <> usiChg
		AND (eStatus = Idle AND eStat = AutoRcpActIdle)  THEN
		CASE p_eNtParamAutoRcpPrecededBy OF
			PrecededBySelf:
				a_tyZ2RcpWr := a_tyCurrZ2Rcp;
			PrecededByF1:
				a_tyMagPropsWr := a_tyMagProps;
		END_CASE
		p_eAct := AutoRcpActWriteRetain;
	END_IF
	IF eStatus = Done AND eStat = AutoRcpActWriteRetain THEN
		usiPrevChg :=  usiChg;
		p_eAct := AutoRcpActIdle;
	END_IF

END_ACTION
```

#### Act_Background2.st - Do Not Change!!!
```iecst
(** 2021-05-18 **)
ACTION Act_Background2:

	CASE p_eNtParamAutoRcpPrecededBy OF
		PrecededBySelf:
			PrecededBySelfBackground2;
		PrecededByF1:
			PrecededByF1Background2;
	END_CASE

END_ACTION
```

#### Act_Action.st - Do Not Change!!!
```iecst
(** 2021-08-01 **)
ACTION Act_Action:

	//Reset Error
	IF (eStatus = Error) AND bRstErr THEN
		p_eAct	:= AutoRcpActIdle;
		eStat	:= AutoRcpActIdle;
	END_IF

	//Set p_eAct
	IF eStatus = Idle OR eStatus = Busy OR eStatus = Done THEN
		eStat	:= p_eAct;
	END_IF

END_ACTION
```

#### Act_Main.st - Do Not Change!!!
```iecst
(** 2021-08-01 **)
ACTION Act_Main:

	IF eStatOld <> eStat THEN
		fbDirCreate1(bEn := FALSE);
		fbDirCreate2(bEn := FALSE);

		fbFileRead1(bEn := FALSE);
		fbFileWrite1(bEn := FALSE);
		fbFileRead2(bEn := FALSE);
		fbFileWrite2(bEn := FALSE);

		usiStep			:= 0;
		bFileNotFound	:= FALSE;

		//sStatTxt	:= a_sStatText[eStat];

		eStatOld	:= eStat;

		eStatus		:= Busy;
	END_IF

	//Main
	CASE eStat OF

		AutoRcpActIdle:
			eStatus	:= Idle;

		AutoRcpActCreateDir:
			IF eStatus = Idle OR eStatus = Busy THEN

				eStatus	:= Busy;

				CASE usiStep OF
					0:
						fbDirCreate1(bEn := TRUE);
						IF fbDirCreate1.udiStatus = 0 THEN
							usiStep	:= 1;
						ELSIF fbDirCreate1.udiStatus < 65534 THEN
							eStatus		:= Error;

							IF fbDirCreate1.udiStatus = 1908 THEN
								udiStatus	:= 10000;	//Create User Directory Error
							ELSE
								udiStatus	:= fbDirCreate1.udiStatus;
							END_IF
						END_IF

					1:
						fbDirCreate2(bEn := TRUE);
						IF fbDirCreate2.udiStatus = 0 THEN
							eStatus	:= Done;
						ELSIF fbDirCreate2.udiStatus < 65534 THEN
							eStatus		:= Error;

							IF fbDirCreate2.udiStatus = 1908 THEN
								udiStatus	:= 10001;	//Create Retain Directory Error
							ELSE
								udiStatus	:= fbDirCreate2.udiStatus;
							END_IF
						END_IF

				END_CASE

			END_IF

		AutoRcpActReadRetain:
			IF eStatus = Idle OR eStatus = Busy THEN

				eStatus	:= Busy;

//				fbFileRead1.p_Dest	:= p_udiRetainDataAddr1;
//				fbFileRead1.udiLen	:= p_udiRetainDataLen1;
				fbFileRead1(bEn := TRUE);

				IF fbFileRead1.udiStatus = 0 THEN
					eStatus	:= Done;
					CASE p_eNtParamAutoRcpPrecededBy OF
						PrecededBySelf:
							a_tyZ2RcpWr := a_tyCurrZ2Rcp;
						PrecededByF1:
							a_tyMagPropsWr := a_tyMagProps;
					END_CASE
					bOverWriteMagProperties := TRUE;

				ELSIF fbFileRead1.udiStatus < 65534 THEN
					eStatus	:= Error;

					IF fbFileRead1.udiStatus = 1900 THEN
						udiStatus	:= 10002;	//File Open Error While Reading Retain File
					ELSIF fbFileRead1.udiStatus = 1902 THEN
						udiStatus	:= 10003;	//File Read Error While Reading Retain File
					ELSIF fbFileRead1.udiStatus = 1904 THEN
						udiStatus	:= 10004;	//File Close Error While Reading Retain File
					ELSIF fbFileRead1.udiStatus = 1915 THEN
						eStatus			:= Done;
						bFileNotFound	:= TRUE;
					ELSE
						udiStatus	:= fbFileRead1.udiStatus;
					END_IF
				END_IF

			END_IF

		AutoRcpActWriteRetain:
			IF eStatus = Idle OR eStatus = Busy THEN

				eStatus	:= Busy;

//				fbFileWrite1.p_Src	:= p_udiRetainDataAddr1;
//				fbFileWrite1.udiLen	:= p_udiRetainDataLen1;
				fbFileWrite1(bEn := TRUE);

				IF fbFileWrite1.udiStatus = 0 THEN
					eStatus	:= Done;
				ELSIF fbFileWrite1.udiStatus < 65534 THEN
					eStatus	:= Error;

					IF fbFileWrite1.udiStatus = 1900 THEN
						udiStatus	:= 10005;	//File Open Error While Writing Retain File
					ELSIF fbFileWrite1.udiStatus = 1901 THEN
						udiStatus	:= 10006;	//File Create Error While Writing Retain File
					ELSIF fbFileWrite1.udiStatus = 1903 THEN
						udiStatus	:= 10007;	//File Write Error While Writing Retain File
					ELSIF fbFileWrite1.udiStatus = 1904 THEN
						udiStatus	:= 10008;	//File Close Error While Writing Retain File
					ELSIF fbFileWrite1.udiStatus = 1914 THEN
						udiStatus	:= 10009;	//Directory Does Not Exist While Writing Retain File
					ELSE
						udiStatus	:= fbFileWrite1.udiStatus;
					END_IF
				END_IF

			END_IF

		AutoRcpActReadRetain2:
			IF eStatus = Idle OR eStatus = Busy THEN

				eStatus	:= Busy;

				fbFileRead2(bEn := TRUE);

				IF fbFileRead2.udiStatus = 0 THEN
					eStatus	:= Done;
					tyZ1RcpWr := tyCurrZ1Rcp;
					bOverWriteTravLifProperties := TRUE;
				ELSIF fbFileRead2.udiStatus < 65534 THEN
					eStatus	:= Error;

					IF fbFileRead2.udiStatus = 1900 THEN
						udiStatus	:= 10002;	//File Open Error While Reading Retain File
					ELSIF fbFileRead2.udiStatus = 1902 THEN
						udiStatus	:= 10003;	//File Read Error While Reading Retain File
					ELSIF fbFileRead2.udiStatus = 1904 THEN
						udiStatus	:= 10004;	//File Close Error While Reading Retain File
					ELSIF fbFileRead2.udiStatus = 1915 THEN
						eStatus			:= Done;
						bFileNotFound	:= TRUE;
					ELSE
						udiStatus	:= fbFileRead2.udiStatus;
					END_IF
				END_IF

			END_IF

		AutoRcpActWriteRetain2:
			IF eStatus = Idle OR eStatus = Busy THEN

				eStatus	:= Busy;

				fbFileWrite2(bEn := TRUE);

				IF fbFileWrite2.udiStatus = 0 THEN
					eStatus	:= Done;
				ELSIF fbFileWrite2.udiStatus < 65534 THEN
					eStatus	:= Error;

					IF fbFileWrite2.udiStatus = 1900 THEN
						udiStatus	:= 10005;	//File Open Error While Writing Retain File
					ELSIF fbFileWrite2.udiStatus = 1901 THEN
						udiStatus	:= 10006;	//File Create Error While Writing Retain File
					ELSIF fbFileWrite2.udiStatus = 1903 THEN
						udiStatus	:= 10007;	//File Write Error While Writing Retain File
					ELSIF fbFileWrite2.udiStatus = 1904 THEN
						udiStatus	:= 10008;	//File Close Error While Writing Retain File
					ELSIF fbFileWrite2.udiStatus = 1914 THEN
						udiStatus	:= 10009;	//Directory Does Not Exist While Writing Retain File
					ELSE
						udiStatus	:= fbFileWrite2.udiStatus;
					END_IF
				END_IF

			END_IF

		ELSE
			IF eStatus = Idle OR eStatus = Busy THEN
				eStatus	:= Done;
			END_IF

	END_CASE

END_ACTION
```

#### Act_Main_Disable.st - Do Not Change!!!
```iecst
(** 2020-09-21 **)
ACTION Act_Main_Disable:

	bUSAllow			:= TRUE;
	bDSAllow			:= TRUE;

	usiProdAccDatStep		:= 0;
	usiProdUpdtDatStep		:= 0;
	tyInfoData.sProgNm		:= '';
	tyInfoData.udiCode		:= 0;
	tyInfoData.eSeverity	:= AlmSeverityNA;
	tyInfoData.sAlmMsg		:= '';

	usiMagAccDatStep		:= 0;
	tyInfoData1.sProgNm		:= '';
	tyInfoData1.udiCode		:= 0;
	tyInfoData1.eSeverity	:= AlmSeverityNA;
	tyInfoData1.sAlmMsg		:= '';

	eStatus		:= Idle;
	udiStatus	:= 0;
	bProdRcpErr	:= FALSE;
	bMagRcpErr	:= FALSE;

END_ACTION
```

#### Act_Alarm.st - Do Not Change!!!
```iecst
(** 2019-04-21 **)
ACTION Act_Alarm:

	//Error
	IF EDGEPOS(eStatus = Error) THEN

		tyAlmData.sProgNm		:= p_sProgNm;
		tyAlmData.udiCode		:= udiStatus;
		tyAlmData.eSeverity		:= AlmSeverityError;
		tyAlmData.udiRunTime	:= tyAlmData.udiRunTime + 1;
		tyAlmData.bAlm			:= TRUE;
		tyAlmData.udiModuleNum  := udiModuleNum;
		g_sAutoRcpProgNm		:= p_sProgNm;
		//Get Error Message
		IF tyAlmData.udiCode < 10000 OR tyAlmData.udiCode > 10099 THEN
			tyAlmData.sAlmMsg	:= 'Unknown';
			tyAlmData.sRcyMsg	:= 'Unknown';
		ELSE
			tyAlmData.sAlmMsg	:= a_tyAlmText[tyAlmData.udiCode].sAlmText;
			tyAlmData.sRcyMsg	:= a_tyAlmText[tyAlmData.udiCode].sRcyText;
		END_IF

	ELSIF bRstErr AND (tyAlmData.udiCode <> 0) THEN

		tyAlmData.udiCode	:= 0;
		tyAlmData.eSeverity	:= AlmSeverityNA;
		tyAlmData.sAlmMsg	:= '';
		tyAlmData.sRcyMsg	:= '';
		tyAlmData.bAlm			:= FALSE;
	END_IF

END_ACTION
```

#### InputRef.var - Do Not Change!!!
```iecst
(*2020-08-06*)
(**)
(*General*)
VAR
	p_eAct : REFERENCE TO eAutoRcpAction;
	p_udiRstErr : REFERENCE TO UDINT;
	p_bPrep : REFERENCE TO BOOL;
	p_bEn : REFERENCE TO BOOL;
	p_bDis : REFERENCE TO BOOL;
END_VAR
(**)
(*Configuration*)
VAR
	p_eAWStat : REFERENCE TO eAWAction;
	p_sIPAddr : REFERENCE TO STRING[15];
END_VAR
(**)
(*Input*)
VAR
	p_bNtParamAutoRcpPrep : REFERENCE TO BOOL;
	p_bMcParamAutoRcpDis : REFERENCE TO BOOL;
	p_sMcNm : REFERENCE TO STRING[30];
	p_bAWPrep : REFERENCE TO BOOL;
	p_bAWDis : REFERENCE TO BOOL;
	p_bMnlAccData : REFERENCE TO BOOL;
	p_bSectionLeader : REFERENCE TO BOOL;
	p_sMagRcpNm : REFERENCE TO STRING[30];
	p_diWidthLimit : REFERENCE TO DINT;
	p_bWidth2Prep : REFERENCE TO BOOL;
	p_bUSWidthChkPrep : REFERENCE TO BOOL;
	p_bUSWidthChkEn : REFERENCE TO BOOL;
	p_bUSWidthChkSen : REFERENCE TO BOOL;
	p_bDSWidthChkPrep : REFERENCE TO BOOL;
	p_bDSWidthChkEn : REFERENCE TO BOOL;
	p_bDSWidthChkSen : REFERENCE TO BOOL;
	p_bProdWidthChk : REFERENCE TO BOOL;
	p_bUIProdAccData : REFERENCE TO BOOL;
	p_bUIProdUpdtData : REFERENCE TO BOOL;
	p_bUIMagAccData : REFERENCE TO BOOL;
	p_tyCmpRcp : REFERENCE TO tyBoardProperty;
	p_sCurrMagRcpNm : REFERENCE TO STRING[30];
	p_eTimeStat : REFERENCE TO eTimeAction;
	p_eTimeStatus : REFERENCE TO eFBStatus;
	p_bAccNewRcpCond : REFERENCE TO BOOL;
	p_bUpdtNewRcpCond : REFERENCE TO BOOL;
	p_bAutoUpdtData : REFERENCE TO BOOL;
	p_sInfoMsg : REFERENCE TO STRING[200];
	p_bInternalUse : REFERENCE TO BOOL;
	p_tyInternalReqProdRcp : REFERENCE TO tyProdRcpParam;
	p_eNtParamAutoRcpPrecededBy : REFERENCE TO eAutoRcpPreceded;
	p_bNtParamProjMagAWPrep : REFERENCE TO BOOL;
	p_bNtParamF1ArbitraryType : REFERENCE TO BOOL;
	p_sTCPTopFullMsgRd : REFERENCE TO STRING[80];
	p_sTCPBtmFullMsgRd : REFERENCE TO STRING[80];
	p_bProdRcp0ToptoBtm : REFERENCE TO BOOL;
	p_bHermesBrdAvlDataNewBrdAvl1stZ : REFERENCE TO BOOL;
	pa_tyLinkXMLTableDataBrdAvl1 : REFERENCE TO ARRAY[0..200] OF tyXMLTableDat;
	p_iLinkXMLTableDataBrdAvlTtlIdx1 : REFERENCE TO INT;
	p_usiLinkProdRcpCurrRcpMcMod : REFERENCE TO USINT;
	pa_bMagRej : REFERENCE TO ARRAY[1..3] OF BOOL;
	p_bOpsMagConvUL1AWDone : REFERENCE TO BOOL;
	p_bOpsMagConvUL2AWDone : REFERENCE TO BOOL;
	p_bOpsMagConvUL3AWDone : REFERENCE TO BOOL;
	p_bOpsMagConvUL1SlotUpdtDone : REFERENCE TO BOOL;
	p_bOpsMagConvUL2SlotUpdtDone : REFERENCE TO BOOL;
	p_bOpsMagConvUL3SlotUpdtDone : REFERENCE TO BOOL;
	p_bMcParamAutoRcpBatchIDChgCmp : REFERENCE TO BOOL;
	p_bMcParamAutoRcpIgnoreBtmClr : REFERENCE TO BOOL;
	p_bMcParamAutoRcpIgnoreTopClr : REFERENCE TO BOOL;
	p_bMcParamAutoRcpIgnoreThickns : REFERENCE TO BOOL;
	p_eNtParamAutoRcpParamLmt : REFERENCE TO eAutoRcpLmt;
	p_diNtParamProdRcpMinWidth : REFERENCE TO DINT;
	p_diNtParamProdRcpMaxWidth : REFERENCE TO DINT;
	p_eULMod : REFERENCE TO eULMod;
	p_bNewBrdEnteredCond : REFERENCE TO BOOL;
	p_bOldBrdExitedCond : REFERENCE TO BOOL;
	p_bRlsBrd : REFERENCE TO BOOL;
	p_tyToLeaderProdRcp : REFERENCE TO tyProdRcpParam;
	pa_bInternalReqProdRcpDiff : REFERENCE TO ARRAY[0..3] OF BOOL;
	p_bUpdtProdRcpDiff : REFERENCE TO BOOL;
	p_bRlsBrdProdRcpDiff : REFERENCE TO BOOL;
	p_sProgNm : REFERENCE TO STRING[15];
	p_bNtSettingsLoadDone : REFERENCE TO BOOL;
	p_tOnlineChkDlyTm : REFERENCE TO TIME;
	p_bManual : REFERENCE TO BOOL;
	p_bErr : REFERENCE TO BOOL;
	p_bWarning : REFERENCE TO BOOL;
	p_bOps : REFERENCE TO BOOL;
	p_bStandby : REFERENCE TO BOOL;
	p_bDBAOnWOAlign : REFERENCE TO BOOL;
END_VAR
(*weFab*)
VAR
	p_tyMagCmpRcp : REFERENCE TO tyMagProperties;
	p_tyCurrProdRcp : REFERENCE TO tyProdRcpParam;
END_VAR
```

#### Local.var - Do Not Change!!!
```iecst
(*2021-05-18*)
(**)
(*Local Action, State & Status*)
VAR
	eAct : eAutoRcpAction;
	eStatus : eFBStatus := Idle;
	udiStatus : UDINT := 0;
	eStatOld : eAutoRcpAction := AutoRcpActIdle;
	eStat : eAutoRcpAction;
	usiStep : USINT;
END_VAR
(**)
(*Local Alarm*)
VAR
	tyAlmData : tyAlmDat;
	tyInfoData : tyAlmDat;
	tyInfoData1 : tyAlmDat;
	a_tyAlmText : ARRAY[10000..10099] OF tyAlmTxt := [(sAlmText:='Create User Directory Error',sRcyText:='An Error Occurred While Attempting To Create User Directory. Please Contact Nutek For A Possible Solution'),(sAlmText:='Create Retain Directory Error',sRcyText:='An Error Occurred While Attempting To Create Retain Directory. Please Contact Nutek For A Possible Solution'),(sAlmText:='File Open Error While Reading Retain File',sRcyText:='An Error Was Encountered While Trying To Open File. Please Contact Nutek For A Possible Solution.'),(sAlmText:='File Read Error While Reading Retain File',sRcyText:='An Error Was Encountered While Trying To Read File. Please Contact Nutek For A Possible Solution.'),(sAlmText:='File Close Error While Reading Retain File',sRcyText:='An Error Was Encountered While Trying To Close File. Please Contact Nutek For A Possible Solution.'),(sAlmText:='File Open Error While Writing Retain File',sRcyText:='An Error Was Encountered While Trying To Open File. Please Contact Nutek For A Possible Solution.'),(sAlmText:='File Create Error While Writing Retain File',sRcyText:='An Error Was Encountered While Trying To Create File. Please Contact Nutek For A Possible Solution.'),(sAlmText:='File Write Error While Writing Retain File',sRcyText:='An Error Was Encountered While Trying To Write File. Please Contact Nutek For A Possible Solution.'),(sAlmText:='File Close Error While Writing Retain File',sRcyText:='An Error Was Encountered While Trying To Close File. Please Contact Nutek For A Possible Solution.'),(sAlmText:='Directory Does Not Exist While Writing Retain File',sRcyText:='The Directory Does Not Exist. Please Contact Nutek For A Possible Solution.'),3(0),3((0)),(sAlmText:='File Create Error While Writing Config File',sRcyText:='An Error Was Encountered While Trying To Create File. Please Contact Nutek For A Possible Solution.'),(0),(sAlmText:='File Close Error While Writing Config File',sRcyText:='An Error Was Encountered While Trying To Close File. Please Contact Nutek For A Possible Solution.'),11((0)),(sAlmText:='File Open Error While Writing Retain File Lane 2',sRcyText:='An Error Was Encountered While Trying To Open File. Please Contact Nutek For A Possible Solution.'),(0),(sAlmText:='File Open Error While Reading Lane 2 Retain File',sRcyText:='An Error Was Encountered While Trying To Open File. Please Contact Nutek For A Possible Solution.'),(sAlmText:='File Read Error While Reading Lane 2 Retain File',sRcyText:='An Error Was Encountered While Trying To Read File. Please Contact Nutek For A Possible Solution.'),(sAlmText:='File Close Error While Reading Lane 2 Retain File',sRcyText:='An Error Was Encountered While Trying To Close File. Please Contact Nutek For A Possible Solution.'),(sAlmText:='File Open Error While Writing Lane 2 Retain File',sRcyText:='An Error Was Encountered While Trying To Open File. Please Contact Nutek For A Possible Solution.'),(sAlmText:='File Create Error While Writing Lane 2 Retain File',sRcyText:='An Error Was Encountered While Trying To Create File. Please Contact Nutek For A Possible Solution.'),(sAlmText:='File Write Error While Writing Lane 2 Retain File',sRcyText:='An Error Was Encountered While Trying To Write File. Please Contact Nutek For A Possible Solution.'),(sAlmText:='File Close Error While Writing Lane 2 Retain File',sRcyText:='An Error Was Encountered While Trying To Close File. Please Contact Nutek For A Possible Solution.'),(sAlmText:='Directory Does Not Exist While Writing Lane 2 Retain File',sRcyText:='The Directory Does Not Exist. Please Contact Nutek For A Possible Solution.'),2((0)),(sAlmText:='File Open Error While Reading Lane 3 Retain File',sRcyText:='An Error Was Encountered While Trying To Open File. Please Contact Nutek For A Possible Solution.'),(sAlmText:='File Read Error While Reading Lane 3 Retain File',sRcyText:='An Error Was Encountered While Trying To Read File. Please Contact Nutek For A Possible Solution.'),(sAlmText:='File Close Error While Reading Lane 3 Retain File',sRcyText:='An Error Was Encountered While Trying To Close File. Please Contact Nutek For A Possible Solution.'),(sAlmText:='File Open Error While Writing Lane 3 Retain File',sRcyText:='An Error Was Encountered While Trying To Open File. Please Contact Nutek For A Possible Solution.'),(sAlmText:='File Create Error While Writing Lane 3 Retain File',sRcyText:='An Error Was Encountered While Trying To Create File. Please Contact Nutek For A Possible Solution.'),(sAlmText:='File Write Error While Writing Lane 3 Retain File',sRcyText:='An Error Was Encountered While Trying To Write File. Please Contact Nutek For A Possible Solution.'),(sAlmText:='File Close Error While Writing Lane 3 Retain File',sRcyText:='An Error Was Encountered While Trying To Close File. Please Contact Nutek For A Possible Solution.'),(sAlmText:='Directory Does Not Exist While Writing Lane 3 Retain File',sRcyText:='The Directory Does Not Exist. Please Contact Nutek For A Possible Solution.'),2((0)),(sAlmText:='File Open Error While Reading Lane 4 Retain File',sRcyText:='An Error Was Encountered While Trying To Open File. Please Contact Nutek For A Possible Solution.'),(sAlmText:='File Read Error While Reading Lane 4 Retain File',sRcyText:='An Error Was Encountered While Trying To Read File. Please Contact Nutek For A Possible Solution.'),(sAlmText:='File Close Error While Reading Lane 4 Retain File',sRcyText:='An Error Was Encountered While Trying To Close File. Please Contact Nutek For A Possible Solution.'),(sAlmText:='File Open Error While Writing Lane 4 Retain File',sRcyText:='An Error Was Encountered While Trying To Open File. Please Contact Nutek For A Possible Solution.'),(sAlmText:='File Create Error While Writing Lane 4 Retain File',sRcyText:='An Error Was Encountered While Trying To Create File. Please Contact Nutek For A Possible Solution.'),(sAlmText:='File Write Error While Writing Lane 4 Retain File',sRcyText:='An Error Was Encountered While Trying To Write File. Please Contact Nutek For A Possible Solution.'),(sAlmText:='File Close Error While Writing Lane 4 Retain File',sRcyText:='An Error Was Encountered While Trying To Close File. Please Contact Nutek For A Possible Solution.'),(sAlmText:='Directory Does Not Exist While Writing Lane 4 Retain File',sRcyText:='The Directory Does Not Exist. Please Contact Nutek For A Possible Solution.'),40((0))];
END_VAR
(**)
(*Local Output*)
VAR
	bUSAllow : BOOL;
	bDSAllow : BOOL;
	tyLeaderInfo : tyLFLeaderInfo;
END_VAR
(**)
(*Local Input*)
VAR
	udiRstErr : UDINT := 0;
	bPrep : BOOL := TRUE;
	bEn : BOOL := TRUE;
	bDis : BOOL := FALSE;
	sIPAddr : STRING[15] := '192.168.0.100';
	sMcNm : STRING[30];
	bAWPrep : BOOL := TRUE;
	bAWDis : BOOL;
	bMnlAccData : BOOL;
	bSectionLeader : BOOL;
	sMagRcpNm : STRING[30];
	diWidthLimit : DINT;
	bWidth2Prep : BOOL;
	bUSWidthChkPrep : BOOL;
	bBffrMagRemoved : BOOL;
	bUSWidthChkEn : BOOL;
	bUSWidthChkSen : BOOL;
	bDSWidthChkPrep : BOOL;
	bDSWidthChkEn : BOOL;
	bDSWidthChkSen : BOOL;
	bProdWidthChk : BOOL;
	bUIProdAccData : BOOL;
	bUIProdUpdtData : BOOL;
	bUIMagAccData : BOOL;
	tyCurrProdRcp : tyBoardProperty;
	sCurrMagRcpNm : STRING[30];
	eTimeStat : eTimeAction;
	eTimeStatus : eFBStatus;
	bAccNewRcpCond : BOOL;
	bUpdtNewRcpCond : BOOL;
	bAutoUpdtData : BOOL;
	sInfoMsg : STRING[200];
	bInternalUse : BOOL;
	tyInternalReqProdRcp : tyProdRcpParam;
	bNewBrdEnteredCond : BOOL;
	bOldBrdExitedCond : BOOL;
	bRlsBrd : BOOL;
	tyToLeaderProdRcp : tyProdRcpParam;
	a_bInternalReqProdRcpDiff : ARRAY[0..3] OF BOOL;
	bUpdtProdRcpDiff : BOOL;
	bRlsBrdProdRcpDiff : BOOL;
	sProgNm : STRING[15] := 'Follower';
	bNtSettingsLoadDone : BOOL := TRUE;
	tOnlineChkDlyTm : TIME;
	bManual : BOOL := FALSE;
	bErr : BOOL := FALSE;
	bWarning : BOOL := FALSE;
	bOps : BOOL := FALSE;
	bStandby : BOOL := FALSE;
	eAWStat : eAWAction;
	bFileNotFound : BOOL;
END_VAR
(**)
(*Local*)
VAR
	bRstErr : BOOL;
	udiRstErrOld : UDINT;
	bInitDone : BOOL;
	bInitialDone : BOOL;
	bAutoAccData : BOOL;
	bProdRcpErr : BOOL;
	bMagRcpErr : BOOL;
	bSetTmErr : BOOL;
	bProdAccDataReq : BOOL;
	sReqProdRcpNm : STRING[254];
	diReqProdRcpWidth : DINT;
	bMagAccDataReq : BOOL;
	sReqMagRcpNm : STRING[30];
	usiProdAccDatStep : USINT;
	usiMagAccDatStep : USINT;
	usiProdUpdtDatStep : USINT;
	tyRlsBrdProdRcpNm : tyProdRcpParam;
	bNewBrdEntered : BOOL;
	bOldBrdExited : BOOL;
	i : INT;
	bFollowerInfo : BOOL;
	bDBAOnWOAlign : BOOL;
	tyProRcpCurrRcp : USINT;
	ProdRcpAct : USINT;
	a_bBufferMagPresent : ARRAY[1..3] OF BOOL := [3(FALSE)];
	a_bForceChgWidthIfSameRcp : ARRAY[1..4] OF BOOL;
	a_bMagAWWidthDiff : ARRAY[1..4] OF BOOL := [4(FALSE)];
	a_tyBffrStat : ARRAY[1..4] OF tyBffrStat := [4((0))];
	a_sortedMagPriority : ARRAY[1..4] OF USINT;
	a_udiMagAllwMagPresentTm : ARRAY[1..4] OF UDINT;
	x : INT;
	ii : INT;
	jj : INT;
	kk : INT;
	usiMag : USINT;
	bCheckNeedMtyMag : BOOL;
	bTravLifWidthDiffBlk : BOOL;
	a_bMagChangOverBlk : ARRAY[1..4] OF BOOL;
	a_bAllwChangeWidth : ARRAY[1..4] OF BOOL;
	a_bAllwChangeSlot : ARRAY[1..4] OF BOOL;
	a_udiMagAllwGo : ARRAY[1..4] OF UDINT;
	bForceExitMag : BOOL;
	udiMagAllwGo : ARRAY[1..4] OF UDINT;
	a_bCheckDifferent : ARRAY[1..4] OF BOOL;
	udiModuleNum : UDINT := 7201;
	usiPrevChg2 : USINT;
	usiChg2 : USINT;
	usiPrevChg : USINT;
	usiChg : USINT;
	iChgOvrCntr : INT;
END_VAR
(*local variable*)
VAR
	bTest : BOOL;
	bTest2 : BOOL;
	bMagWriteRetain : BOOL;
	bInitializedFollower1Done : BOOL;
	bOverWriteMagProperties : BOOL;
	bOverWriteTravLifProperties : BOOL;
	bZ1AccNewRcpCondition : BOOL;
	bZ2AccNewRcpCondition : BOOL;
	diRequestedMinSlt : DINT := 3;
	diRequestedGapToMaxSlt : DINT;
	bHermesBAAccpt : BOOL;
	bHermesBFAccpt : BOOL;
	tyHermesBAAccpt : tyHermesBoardAvailable;
	tyHermesBFAccpt : tyHermesBoardForecast;
END_VAR
(*Local Variable for calculation*)
VAR
	rMinslt : REAL;
	rMaxslt : REAL;
	rPitch : REAL;
	rNumInterval : REAL;
	diCalcedPitch : DINT;
	diCalcedMax : DINT;
	diCalcedMin : DINT;
	diModulus : DINT;
	sProdtypeID : STRING[254];
	diProdWidth : DINT;
	eULMode : eULMod;
END_VAR
(*Rcp Property*)
VAR
	tyCurrReqRcp : tyBoardProperty;
	tyCurrZ1Rcp : tyBoardProperty; (*For Conveyor*)
	a_tyCurrZ2Rcp : ARRAY[1..4] OF tyBoardProperty; (*Mag1*)
END_VAR
(*Write Rcp*)
VAR
	tyZ1RcpWr : tyBoardProperty; (*For Conveyor*)
	a_tyZ2RcpWr : ARRAY[1..4] OF tyBoardProperty; (*Mag1*)
END_VAR
(*from Z2RcpWr to Conveted Mag Properties*)
VAR
	diTravLifWidth : DINT;
	a_tyMagProps : ARRAY[1..4] OF tyMagProperties;
END_VAR
(*Save Magazine Rcp*)
VAR
	fbDirCreate1 : fbDirCreate;
	fbDirCreate2 : fbDirCreate;
	fbFileRead1 : fbFileFullRead;
	fbFileRead2 : fbFileFullRead;
	fbFileRead3 : fbFileFullRead;
	fbFileWrite1 : fbFileFullWrite;
	fbFileWrite2 : fbFileFullWrite;
	fbFileWrite3 : fbFileFullWrite;
	fbParseBrdAvlExternal : fbHermesParseXMLTable;
END_VAR
(*WeFab*)
VAR
	tyCurrReqMagRcp : tyMagProperties;
	a_tyMagPropsWr : ARRAY[1..4] OF tyMagProperties;
END_VAR
```

### MagConv.typ - Change By Project
```iecst
(*2019-05-28*)
(**)
(*Action*)

TYPE
	eMagConvAction :
		(
		MagConvActIdle,
		MagConvActInit,
		MagConvActInitStopClp,
		MagConvActInitClpStop,
		MagConvActEnt,
		MagConvActEntStopClp,
		MagConvActEntClpStop,
		MagConvActPreExit,
		MagConvActPreExitClpr,
		MagConvActExit,
		MagConvActExit1,
		MagConvActExitClpr,
		MagConvActExit1Clpr,
		MagConvActClprSetAll,
		MagConvActClprRstAll,
		MagConvActClprSetClamp,
		MagConvActClprSetUnclamp,
		MagConvActClprClamp,
		MagConvActClprUnclamp,
		MagConvActStop,
		MagConvActStopClpr,
		MagConvActSetMtrSigOnOrLToR,
		MagConvActSetMtrDirOrRToL,
		MagConvActRstMtrSigOnOrLToR,
		MagConvActRstMtrDirOrRToL,
		MagConvActSetMtrAll,
		MagConvActRstMtrAll
		);
END_TYPE

(**)
```

### InMagConv.var - Change By Project
```iecst
(*2019-03-25*)
(**)
(*Action & State & Status*)
VAR
	p_InMagConvStat : UDINT;
	p_InMagConvStatus : UDINT;
	p_InMagConvStatTxt : UDINT;
END_VAR
(**)
(*Alarm*)
VAR
	p_InMagConvAlmData : UDINT;
END_VAR
(**)
(*Output*)
VAR
	p_InMagConvHvMag : UDINT;
	p_InMagConvMtrSigOnOrLToR : UDINT;
	p_InMagConvMtrDirOrRToL : UDINT;
	p_InMagConvClprClampCtrl : UDINT;
	p_InMagConvClprTwoOutputControl : UDINT;
END_VAR
```

### Program Logical/MagConv_TopBtm/InMagConv (IEC) - 1.00.0 - NtConv v5.00.0 , NtPneu v5.00.0

#### InputRef_Link.var
```iecst
(*2019-04-09*)
(**)
VAR
	p_bLinkOpsRun : REFERENCE TO BOOL;
END_VAR
(**)
VAR
	p_bLinkDISafetyRlySig : REFERENCE TO BOOL;
	p_bLinkOpsInitULDStepInitDone : REFERENCE TO BOOL;
	p_bLinkInMagConvMidSen : REFERENCE TO BOOL;
	p_bLinkInMagConvExtSen : REFERENCE TO BOOL;
	p_bLinkLifterLmtSW : REFERENCE TO BOOL;
	fbLeftSenOnChk : TON;
	p_bLinkOpsInMagConvStepEntToMid : REFERENCE TO BOOL;
END_VAR
```

#### Local.var
```iecst
(*2019-05-28*)
(**)
(*Local Action, State & Status*)
VAR
	eAct : eMagConvAction := MagConvActIdle;
	eStat : eMagConvAction := MagConvActIdle;
	eStatus : eFBStatus := Idle;
	udiStatus : UDINT := 0;
	sStatTxt : STRING[200] := '';
	a_sStatText : ARRAY[0..50] OF STRING[200] := ['Idling','Initializing','Initializing With Stop Then Clamper','Initializing With Clamper Then Stop','Entering Board','Entering Board With Stop Then Clamper','Entering Board With Clamper Then Stop','Pre-Exiting Board','Pre-Exiting Board With Clamper',2('Exiting Board'),2('Exiting Board With Clamper'),'Clamper Setting All Control','Clamper Resetting All Control','Clamper Setting Clamp','Clamper Setting Unclamp','Clamper Clamp','Clampler Unclamp','Stopping','Stopping With Clamper','Turning On Motor Signal','Turning On Motor Direction','Turning Off Motor Signal','Turning Off Motor Direction','Turning On All Motor Output','Turning Off All Motor Output',24('')];
END_VAR
(**)
(*Local Alarm*)
VAR
	tyAlmData : tyAlmDat;
	a_tyAlmText : ARRAY[10000..10099] OF tyAlmTxt := [(sAlmText:='Magazine Detected But Not Present At Outlet Sensor (L - R) While Magazine Conveyor Initial',sRcyText:='Operation Interrupted By Undetected Magazine. Adjusting The Magazine Or Remove The Present Magazine To Resume Operation.'),(sAlmText:='Magazine Detected But Not Present At Outlet Sensor (R - L) While Magazine Conveyor Initial',sRcyText:='Operation Interrupted By Undetected Magazine. Adjusting The Magazine Or Remove The Present Magazine To Resume Operation.'),(sAlmText:='Clamper Clamp Sensor Off Time Out In Unclamp Check While Conveyor Initial With Clamper',sRcyText:='Sensor Timeout Expired Before Operation Completed. Sensor Operation Is Abnormal. Solve The Error To Resume Operation.'),(sAlmText:='Clamper Unclamp Sensor On Time Out In Unclamp Check While Conveyor Initial With Clamper',sRcyText:='Sensor Timeout Expired Before Operation Completed. Sensor Operation Is Abnormal. Solve The Error To Resume Operation.'),(sAlmText:='Clamper Unclamp Safety Sensor Error In Unclamp Check While Conveyor Initial With Clamper',sRcyText:='Safety System Has Been Triggered. All Operations Are Disable. Remove the Obstacle That Triggered The Safety Interlock To Resume Operation.'),(sAlmText:='Magazine Detected But Not Present At Outlet Sensor (L - R) While Conveyor Initial With Clamper',sRcyText:='Operation Interrupted By Undetected Magazine. Adjusting The Magazine Or Remove The Present Magazine To Resume Operation.'),(sAlmText:='Magazine Detected But Not Present At Outlet Sensor (R - L) While Conveyor Initial With Clamper',sRcyText:='Operation Interrupted By Undetected Magazine. Adjusting The Magazine Or Remove The Present Magazine To Resume Operation.'),(sAlmText:='Clamper Clamp Sensor On Time Out In Clamp Check While Conveyor Initial With Clamper',sRcyText:='Sensor Timeout Expired Before Operation Completed. Sensor Operation Is Abnormal. Solve The Error To Resume Operation.'),(sAlmText:='Clamper Unclamp Sensor Off Time Out In Clamp Check While Conveyor Initial With Clamper',sRcyText:='Sensor Timeout Expired Before Operation Completed. Sensor Operation Is Abnormal. Solve The Error To Resume Operation.'),(sAlmText:='Clamper Clamp Safety Sensor Error In Clamp Check While Conveyor Initial With Clamper',sRcyText:='Safety System Has Been Triggered. All Operations Are Disable. Remove the Obstacle That Triggered The Safety Interlock To Resume Operation.'),(sAlmText:='Clamper Clamp Sensor On Time Out In Clamp Check While Conveyor Enter With Clamper',sRcyText:='Sensor Timeout Expired Before Operation Completed. Sensor Operation Is Abnormal. Solve The Error To Resume Operation.'),(sAlmText:='Clamper Unclamp Sensor Off Time Out In Clamp Check While Conveyor Enter With Clamper',sRcyText:='Sensor Timeout Expired Before Operation Completed. Sensor Operation Is Abnormal. Solve The Error To Resume Operation.'),(sAlmText:='Clamper Clamp Safety Sensor Error In Clamp Check While Conveyor Enter With Clamper',sRcyText:='Safety System Has Been Triggered. All Operations Are Disable. Remove the Obstacle That Triggered The Safety Interlock To Resume Operation.'),(sAlmText:='Clamper Clamp Sensor Off Time Out In Unclamp Check While Conveyor Exit With Clamper',sRcyText:='Sensor Timeout Expired Before Operation Completed. Sensor Operation Is Abnormal. Solve The Error To Resume Operation.'),(sAlmText:='Clamper Unclamp Sensor On Time Out In Unclamp Check While Conveyor Exit With Clamper',sRcyText:='Sensor Timeout Expired Before Operation Completed. Sensor Operation Is Abnormal. Solve The Error To Resume Operation.'),(sAlmText:='Clamper Unclamp Safety Sensor Error In Unclamp Check While Conveyor Exit With Clamper',sRcyText:='Safety System Has Been Triggered. All Operations Are Disable. Remove the Obstacle That Triggered The Safety Interlock To Resume Operation.'),(sAlmText:='Clamper Clamp Sensor On Time Out In Clamp Check While Clamper Clamp',sRcyText:='Sensor Timeout Expired Before Operation Completed. Sensor Operation Is Abnormal. Solve The Error To Resume Operation.'),(sAlmText:='Clamper Unclamp Sensor Off Time Out In Clamp Check While Clamper Clamp',sRcyText:='Sensor Timeout Expired Before Operation Completed. Sensor Operation Is Abnormal. Solve The Error To Resume Operation.'),(sAlmText:='Clamper Clamp Safety Sensor Error In Clamp Check While Clamper Clamp',sRcyText:='Safety System Has Been Triggered. All Operations Are Disable. Remove the Obstacle That Triggered The Safety Interlock To Resume Operation.'),(sAlmText:='Clamper Clamp Sensor Off Time Out In Unclamp Check While Clamper Unclamp',sRcyText:='Sensor Timeout Expired Before Operation Completed. Sensor Operation Is Abnormal. Solve The Error To Resume Operation.'),(sAlmText:='Clamper Unclamp Sensor On Time Out In Unclamp Check While Clamper Unclamp',sRcyText:='Sensor Timeout Expired Before Operation Completed. Sensor Operation Is Abnormal. Solve The Error To Resume Operation.'),(sAlmText:='Clamper Unclamp Safety Sensor Error In Unclamp Check While Clamper Unclamp',sRcyText:='Safety System Has Been Triggered. All Operations Are Disable. Remove the Obstacle That Triggered The Safety Interlock To Resume Operation.'),(sAlmText:='Clamper Clamp Sensor Off Time Out In Unclamp Check While Stop With Clamper',sRcyText:='Sensor Timeout Expired Before Operation Completed. Sensor Operation Is Abnormal. Solve The Error To Resume Operation.'),(sAlmText:='Clamper Unclamp Sensor On Time Out In Unclamp Check While Stop With Clamper',sRcyText:='Sensor Timeout Expired Before Operation Completed. Sensor Operation Is Abnormal. Solve The Error To Resume Operation.'),(sAlmText:='Clamper Unclamp Safety Sensor Error In Unclamp Check While Stop With Clamper',sRcyText:='Safety System Has Been Triggered. All Operations Are Disable. Remove the Obstacle That Triggered The Safety Interlock To Resume Operation.'),(sAlmText:='Clamper Clamp Sensor Off Time Out In Unclamp Check While Conveyor Exit With Clamper',sRcyText:='Sensor Timeout Expired Before Operation Completed. Sensor Operation Is Abnormal. Solve The Error To Resume Operation.'),(sAlmText:='Clamper Unclamp Sensor On Time Out In Unclamp Check While Conveyor Exit With Clamper',sRcyText:='Sensor Timeout Expired Before Operation Completed. Sensor Operation Is Abnormal. Solve The Error To Resume Operation.'),(sAlmText:='Clamper Unclamp Safety Sensor Error In Unclamp Check While Conveyor Exit With Clamper',sRcyText:='Safety System Has Been Triggered. All Operations Are Disable. Remove the Obstacle That Triggered The Safety Interlock To Resume Operation.'),2((sAlmText:='Transfer In Time Out While Entering Magazine',sRcyText:='Timeout Expired Before Operation Completed. Transmission Abnormal. Remove the Obstacle (If Exists) To Resume Operation.')),(sAlmText:='Transfer Out Time Out While Exiting Magazine',sRcyText:='Timeout Expired Before Operation Completed. Transmission Abnormal. Remove the Obstacle (If Exists) To Resume Operation.'),(sAlmText:='Transfer Out Time Out While Conveyor Exit With Clamper',sRcyText:='Timeout Expired Before Operation Completed. Transmission Abnormal. Remove the Obstacle (If Exists) To Resume Operation.'),(sAlmText:='Transfer Out Time Out While Exiting Magazine',sRcyText:='Timeout Expired Before Operation Completed. Transmission Abnormal. Remove the Obstacle (If Exists) To Resume Operation.'),(sAlmText:='Transfer Out Time Out While Conveyor Exit With Clamper',sRcyText:='Timeout Expired Before Operation Completed. Transmission Abnormal. Remove the Obstacle (If Exists) To Resume Operation.'),(sAlmText:='Clamper Clamp Sensor On Time Out In Clamp Check While Conveyor Enter With Clamper',sRcyText:='Sensor Timeout Expired Before Operation Completed. Sensor Operation Is Abnormal. Solve The Error To Resume Operation.'),(sAlmText:='Clamper Unclamp Sensor Off Time Out In Clamp Check While Conveyor Enter With Clamper',sRcyText:='Sensor Timeout Expired Before Operation Completed. Sensor Operation Is Abnormal. Solve The Error To Resume Operation.'),(sAlmText:='Clamper Clamp Safety Sensor Error In Clamp Check While Conveyor Enter With Clamper',sRcyText:='Safety System Has Been Triggered. All Operations Are Disable. Remove the Obstacle That Triggered The Safety Interlock To Resume Operation.'),(sAlmText:='Transfer In Time Out While Entering Magazine',sRcyText:='Timeout Expired Before Operation Completed. Transmission Abnormal. Remove the Obstacle (If Exists) To Resume Operation.'),(sAlmText:='Clamper Clamp Sensor Off Time Out In Unclamp Check While Conveyor Initial With Clamper',sRcyText:='Sensor Timeout Expired Before Operation Completed. Sensor Operation Is Abnormal. Solve The Error To Resume Operation.'),(sAlmText:='Clamper Unclamp Sensor On Time Out In Unclamp Check While Conveyor Initial With Clamper',sRcyText:='Sensor Timeout Expired Before Operation Completed. Sensor Operation Is Abnormal. Solve The Error To Resume Operation.'),(sAlmText:='Clamper Unclamp Safety Sensor Error In Unclamp Check While Conveyor Initial With Clamper',sRcyText:='Safety System Has Been Triggered. All Operations Are Disable. Remove the Obstacle That Triggered The Safety Interlock To Resume Operation.'),(sAlmText:='Magazine Detected But Not Present At Outlet Sensor (L - R) While Conveyor Initial With Clamper',sRcyText:='Operation Interrupted By Undetected Magazine. Adjusting The Magazine Or Remove The Present Magazine To Resume Operation.'),(sAlmText:='Magazine Detected But Not Present At Outlet Sensor (R - L) While Conveyor Initial With Clamper',sRcyText:='Operation Interrupted By Undetected Magazine. Adjusting The Magazine Or Remove The Present Magazine To Resume Operation.'),(sAlmText:='Clamper Clamp Sensor On Time Out In Clamp Check While Conveyor Initial With Clamper',sRcyText:='Sensor Timeout Expired Before Operation Completed. Sensor Operation Is Abnormal. Solve The Error To Resume Operation.'),(sAlmText:='Clamper Unclamp Sensor Off Time Out In Clamp Check While Conveyor Initial With Clamper',sRcyText:='Sensor Timeout Expired Before Operation Completed. Sensor Operation Is Abnormal. Solve The Error To Resume Operation.'),(sAlmText:='Clamper Clamp Safety Sensor Error In Clamp Check While Conveyor Initial With Clamper',sRcyText:='Safety System Has Been Triggered. All Operations Are Disable. Remove the Obstacle That Triggered The Safety Interlock To Resume Operation.'),(sAlmText:='Magazine Not Detected While Pre-Exiting Magazine',sRcyText:='Operation Interrupted By Undetected Magazine. Adjusting The Magazine Or Remove The Present Magazine To Resume Operation.'),53((0))];
END_VAR
(**)
(*Local Output*)
VAR
	bHvMag : BOOL := FALSE;
	bMtrSigOnOrLToR : BOOL := FALSE;
	bMtrDirOrRToL : BOOL := FALSE;
	bClprClampCtrl : BOOL;
	bClprTwoOutputControl : BOOL := FALSE;
END_VAR
(**)
(*Local Input*)
VAR
	udiRstErr : UDINT := 0;
	bPrep : BOOL := TRUE;
	bEn : BOOL := TRUE;
	bDis : BOOL := FALSE;
	bManual : BOOL := FALSE;
	bOnDirMod : BOOL := FALSE;
	diInitTm : DINT := 10000;
	tMtrOffDlyTm : TIME := T#0S;
	diTxInTimeOut : DINT := 10000;
	diTxOutTimeOut : DINT := 10000;
	eDirection : eConvDir := ConvDirLToR;
	bLeftSen : BOOL := FALSE;
	bRightSen : BOOL := FALSE;
	bClprClampSen : BOOL := FALSE;
	bClprUnclampSen : BOOL := FALSE;
	bClprClampSafetySen : BOOL := TRUE;
	bClprUnclampSafetySen : BOOL := TRUE;
	sProgNm : STRING[15] := 'MagConv';
	tClprClampTO : TIME := T#20s;
	tClprUnclampTO : TIME := T#20s;
	bNtSettingsLoadDone : BOOL := TRUE;
END_VAR
(**)
(*Local*)
VAR
	bRstErr : BOOL;
	udiRstErrOld : UDINT;
	bInitDone : BOOL;
	bInitialDone : BOOL;
	bReachEnd : BOOL;
	usiStep : USINT;
	eStatOld : eMagConvAction := MagConvActIdle;
	fbInit : fbConvSenToSenTm;
	fbEnt : fbConvSenToSen;
	fbPreExit : fbConvSenToSenTm;
	fbExit : fbConvSenToSenOff;
	fbExit1 : fbConvSenToSenOff1;
	fbStop : fbConvMtrOff;
	fbClprClampChk : fbPneuExtRetSenExtChk;
	fbClprUnclampChk : fbPneuExtRetSenRetChk;
	fbClprDlyTm : TON;
	udiModuleNum : UDINT := 1801;
END_VAR
```

#### Act_InitGlobal.st
```iecst
(** 2019-04-09 **)
ACTION Act_InitGlobal:

	(* Always Change If Project Change *)

	//Pass Data To Links
	p_bLinkOpsRun ACCESS p_OpsRun;

	p_bLinkDISafetyRlySig ACCESS p_DISafetyRlySig;
	p_bLinkOpsInitULDStepInitDone ACCESS p_OpsLifMagULStepInitDone1;
	p_bLinkInMagConvMidSen ACCESS p_DIInMagConvMidSen;
	p_bLinkInMagConvExtSen ACCESS p_DIInMagConvExtSen;
	p_bLinkLifterLmtSW ACCESS p_DILifterLmtSW;
	p_bLinkOpsInMagConvStepEntToMid ACCESS p_OpsInMagConvStepEntToMid;

	//Pass Data To Internal Use
	p_udiRstErr ACCESS p_RstErrReset;
	p_bManual ACCESS p_UIMnlMod;
	p_bOnDirMod ACCESS p_NtParamInMagConvOnDirMod;
	p_tMtrOffDlyTm ACCESS p_NtParamInMagConvMtrOffDlyTm;
	p_diInitTm ACCESS p_McParamInMagConvRunTmOut;
	p_diTxInTimeOut ACCESS p_McParamInMagConvRunTmOut;
	p_diTxOutTimeOut ACCESS p_McParamInMagConvRunTmOut;
	//p_bRightSen ACCESS p_DIInMagConvMidSen;
	p_eDirection ACCESS p_NtParamProjInMagConvDir;
	p_sProgNm ACCESS p_NtParamInMagConvProgNm;
	p_bNtSettingsLoadDone ACCESS p_StartupNtSettingsLoadDone;

	(* Always Change If Project Change *)

END_ACTION
```

#### Act_Link.st
```iecst
(** 2019-03-29 **)
ACTION Act_Link:
	//InMag unloader -> R-L
	IF p_eAct = MagConvActInit OR p_eAct = MagConvActEnt THEN
		IF p_bLinkOpsInMagConvStepEntToMid THEN
			p_bRightSen ACCESS p_DIInMagConvEntSen;
			p_bLeftSen		:= p_bLinkInMagConvMidSen;
		ELSE
			p_bRightSen ACCESS p_DIInMagConvMidSen;
			p_bLeftSen		:= p_bLinkInMagConvExtSen;
		END_IF

	//	p_bRightSen ACCESS p_DIInMagConvMidSen;
	ELSIF p_eAct = MagConvActExit THEN
		p_bLeftSen		:= p_bLinkLifterLmtSW = FALSE;
		p_bRightSen ACCESS p_DIInMagConvMidSen;
	ELSE
		p_bRightSen ACCESS p_DIInMagConvMidSen;
	END_IF

	IF EDGEPOS(eStatus = Error) THEN
		bMtrSigOnOrLToR	:= FALSE;
		bMtrDirOrRToL	:= FALSE;
	END_IF

END_ACTION
```

#### Act_LinkAction.st
```iecst
(** 2019-04-09 **)
ACTION Act_LinkAction:

	IF p_bLinkOpsRun = TRUE AND p_OpsInMagConvAct <> 0 THEN
//		IF p_bLinkOpsInitULDStepInitDone = FALSE THEN
//			p_eAct ACCESS p_OpsLifMagULInMagConvAct;
//		ELSE
			p_eAct ACCESS p_OpsInMagConvAct;
//		END_IF
	ELSIF p_bManual = TRUE THEN
		p_eAct ACCESS p_UIInMagConvAct;
	ELSE
		p_eAct ACCESS ADR(eAct);
	END_IF

END_ACTION
```

#### Init.st
```iecst
(** 2019-03-25 **)
PROGRAM _INIT

	(* Always Change If Project Change *)

	//Pass Address To Global Address For External Use
	//Action, State & Status
	p_InMagConvStat		:= ADR(eStat);
	p_InMagConvStatus	:= ADR(eStatus);
	p_InMagConvStatTxt	:= ADR(sStatTxt);

	//Alarm
	p_InMagConvAlmData	:= ADR(tyAlmData);

	//Output
	p_InMagConvHvMag				:= ADR(bHvMag);
	p_InMagConvMtrSigOnOrLToR		:= ADR(bMtrSigOnOrLToR);
	p_InMagConvMtrDirOrRToL			:= ADR(bMtrDirOrRToL);

	p_InMagConvClprClampCtrl		:= ADR(bClprClampCtrl);
	p_InMagConvClprTwoOutputControl	:= ADR(bClprTwoOutputControl);

	(* Always Change If Project Change *)

END_PROGRAM
```

### OutMagConv.var - Change By Project
```iecst
(*2019-03-25*)
(**)
(*Action & State & Status*)
VAR
	p_OutMagConvStat : UDINT;
	p_OutMagConvStatus : UDINT;
	p_OutMagConvStatTxt : UDINT;
END_VAR
(**)
(*Alarm*)
VAR
	p_OutMagConvAlmData : UDINT;
END_VAR
(**)
(*Output*)
VAR
	p_OutMagConvHvMag : UDINT;
	p_OutMagConvMtrSigOnOrLToR : UDINT;
	p_OutMagConvMtrDirOrRToL : UDINT;
	p_OutMagConvClprClampCtrl : UDINT;
	p_OutMagConvClprTwoOutControl : UDINT;
END_VAR
```

### Program Logical/MagConv_TopBtm/OutMagConv (IEC) - 1.00.0 - NtConv v5.00.0 , NtPneu v5.00.0

#### InputRef_Link.var
```iecst
(*2019-04-09*)
(**)
VAR
	p_bLinkOpsRun : REFERENCE TO BOOL;
END_VAR
(**)
VAR
	p_bLinkDISafetyRlySig : REFERENCE TO BOOL;
	fbOutMagConvStopTm : TON;
	bTmr : BOOL;
	p_tyLinkDI : REFERENCE TO tyDigitalInputSettings;
	p_bLinkOpsInitULDStepInitDone : REFERENCE TO BOOL;
	p_bLinkOpsOutMagConStepEntMag : REFERENCE TO BOOL;
	p_bLinkOpsOutMagConStepEntMidMag : REFERENCE TO BOOL;
END_VAR
```

#### Act_InitGlobal.st
```iecst
(** 2019-04-09 **)
ACTION Act_InitGlobal:

	(* Always Change If Project Change *)

	//Pass Data To Link
	p_bLinkOpsRun ACCESS p_OpsRun;

	p_bLinkDISafetyRlySig ACCESS p_DISafetyRlySig;
	p_tyLinkDI ACCESS p_NtParamDISettings;
	p_bLinkOpsInitULDStepInitDone ACCESS p_OpsLifMagULStepInitDone1;
	p_bLinkOpsOutMagConStepEntMag ACCESS p_OpsOutMagConvStepEntMag;
	p_bLinkOpsOutMagConStepEntMidMag ACCESS p_OpsOutMagConvStepEntMidMag;

	//Pass Data To Internal Use
	p_udiRstErr ACCESS p_RstErrReset;
	p_bManual ACCESS p_UIMnlMod;
	p_bOnDirMod ACCESS p_NtParamOutMagConvOnDirMod;
	p_tMtrOffDlyTm ACCESS p_NtParamOutMagConvMtrOffDlyTm;
	p_diInitTm ACCESS p_McParamOutMagConvRunTmOut;
	p_diTxInTimeOut ACCESS p_McParamOutMagConvRunTmOut;
	p_diTxOutTimeOut ACCESS p_McParamOutMagConvRunTmOut;
	p_eDirection ACCESS p_NtParamProjOutMagConvDir;
	p_bLeftSen ACCESS p_DIOutMagConvEntSen;
	p_sProgNm ACCESS p_NtParamOutMagConvProgNm;
	p_bNtSettingsLoadDone ACCESS p_StartupNtSettingsLoadDone;

	(* Always Change If Project Change *)

END_ACTION
```

#### Act_InitLocal.st
```iecst
(** 2019-03-25 **)
ACTION Act_InitLocal:

	//Input Reference Link To Local Variable
	p_eAct ACCESS ADR(eAct);
	p_udiRstErr ACCESS ADR(udiRstErr);
	p_bPrep ACCESS ADR(bPrep);
	p_bEn ACCESS ADR(bEn);
	p_bDis ACCESS ADR(bDis);

	p_bManual ACCESS ADR(bManual);
	p_bOnDirMod ACCESS ADR(bOnDirMod);
	p_diInitTm ACCESS ADR(diInitTm);
	p_tMtrOffDlyTm ACCESS ADR(tMtrOffDlyTm);
	p_diTxInTimeOut ACCESS ADR(diTxInTimeOut);
	p_diTxOutTimeOut ACCESS ADR(diTxOutTimeOut);
	p_eDirection ACCESS ADR(eDirection);
	p_sProgNm ACCESS ADR(sProgNm);
	p_tClprClampTO ACCESS ADR(tClprClampTO);
	p_tClprUnclampTO ACCESS ADR(tClprUnclampTO);
	p_bNtSettingsLoadDone ACCESS ADR(bNtSettingsLoadDone);
	p_bLeftSen ACCESS ADR(bLeftSen);
	p_bRightSen ACCESS ADR(bRightSen);
	p_bClprClampSen ACCESS ADR(bClprClampSen);
	p_bClprUnclampSen ACCESS ADR(bClprUnclampSen);
	p_bClprClampSafetySen ACCESS ADR(bClprClampSafetySen);
	p_bClprUnclampSafetySen ACCESS ADR(bClprUnclampSafetySen);

END_ACTION
```

#### Act_Link.st
```iecst
(** 2019-03-29 **)
ACTION Act_Link:

	IF p_tyLinkDI.diOutMagConvExtSen = 0 THEN
		IF EDGENEG (p_bLeftSen) AND (eStat = MagConvActEnt) THEN
			bTmr := TRUE;
		END_IF

		IF bTmr	= TRUE THEN
			fbOutMagConvStopTm(IN := TRUE, PT:=T#3500ms);

			IF fbOutMagConvStopTm.Q THEN
				fbOutMagConvStopTm(IN:=FALSE);

				p_bRightSen := TRUE;
				bTmr		:= FALSE;
			END_IF
		END_IF

		IF (eStat = MagConvActEnt AND eStatus = Done) THEN
			p_bRightSen		:= FALSE;
		END_IF

	ELSIF p_bLinkOpsOutMagConStepEntMag THEN 	//add
		p_bRightSen ACCESS p_DIOutMagConvExtSen;
	ELSIF p_bLinkOpsOutMagConStepEntMidMag THEN //add
		p_bRightSen ACCESS p_DIOutMagConvMidSen;
	ELSE
		p_bRightSen ACCESS p_DIOutMagConvExtSen;
	END_IF

	IF EDGEPOS(eStatus = Error) THEN
		bMtrSigOnOrLToR	:= FALSE;
		bMtrDirOrRToL	:= FALSE;
	END_IF

END_ACTION
```

#### Act_LinkAction.st
```iecst
(** 2019-04-09 **)
ACTION Act_LinkAction:

	IF p_bLinkOpsRun = TRUE AND p_OpsOutMagConvAct <> 0 THEN
//		IF p_bLinkOpsInitULDStepInitDone = FALSE THEN
//			p_eAct ACCESS p_OpsLifMagULOutMagConvAct;
//		ELSE
			p_eAct ACCESS p_OpsOutMagConvAct;
//		END_IF
	ELSIF p_bManual = TRUE THEN
		p_eAct ACCESS p_UIOutMagConvAct;
	ELSE
		p_eAct ACCESS ADR(eAct);
	END_IF

END_ACTION
```
